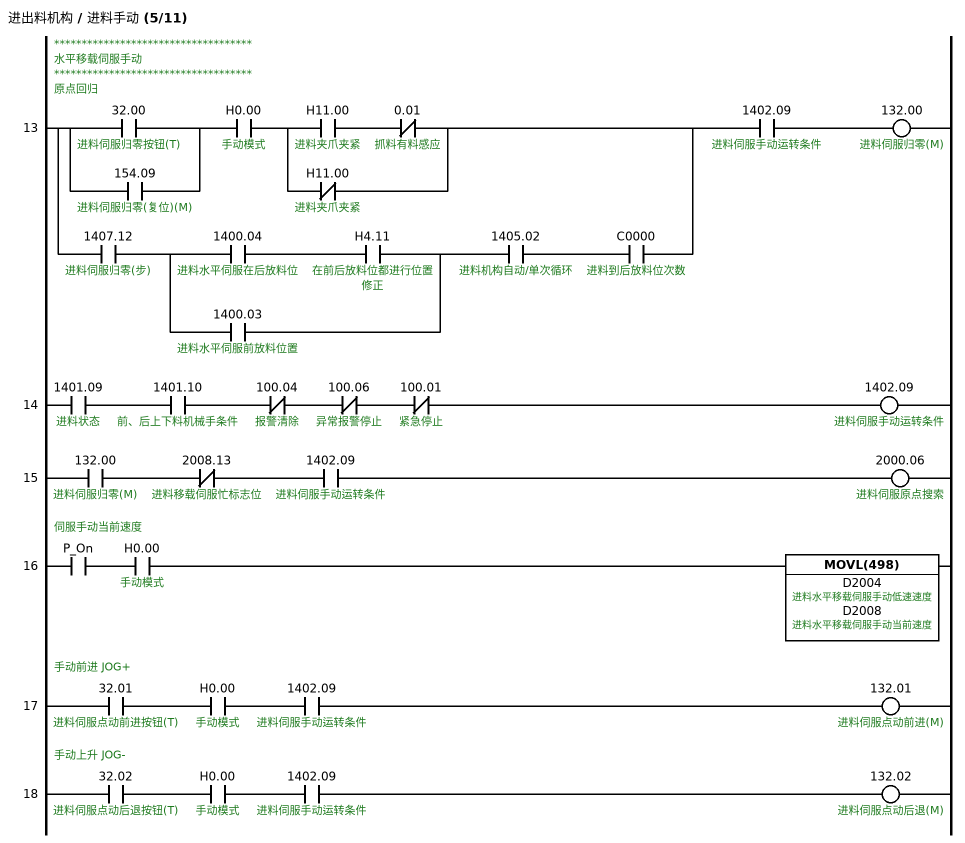
; [picture p72: 进出料机构 / 进料手动, rungs 13-18]
; rung 13: ************************************ / 水平移载伺服手动 / ************************************ / 原点回归
LD 32.00  ; 进料伺服归零按钮(T)
OR 154.09  ; 进料伺服归零(复位)(M)
AND H0.00  ; 手动模式
LD H11.00  ; 进料夹爪夹紧
ANDNOT 0.01  ; 抓料有料感应
ORNOT H11.00  ; 进料夹爪夹紧
ANDLD
LD 1407.12  ; 进料伺服归零(步)
LD 1400.04  ; 进料水平伺服在后放料位
AND H4.11  ; 在前后放料位都进行位置修正
OR 1400.03  ; 进料水平伺服前放料位置
ANDLD
AND 1405.02  ; 进料机构自动/单次循环
AND C0000  ; 进料到后放料位次数
ORLD
AND 1402.09  ; 进料伺服手动运转条件
OUT 132.00  ; 进料伺服归零(M)
; rung 14
LD 1401.09  ; 进料状态
AND 1401.10  ; 前、后上下料机械手条件
ANDNOT 100.04  ; 报警清除
ANDNOT 100.06  ; 异常报警停止
ANDNOT 100.01  ; 紧急停止
OUT 1402.09  ; 进料伺服手动运转条件
; rung 15
LD 132.00  ; 进料伺服归零(M)
ANDNOT 2008.13  ; 进料移载伺服忙标志位
AND 1402.09  ; 进料伺服手动运转条件
OUT 2000.06  ; 进料伺服原点搜索
; rung 16: 伺服手动当前速度
LD P_On
AND H0.00  ; 手动模式
MOVL(498) D2004 D2008  ; 进料水平移载伺服手动低速速度, 进料水平移载伺服手动当前速度
; rung 17: 手动前进 JOG+
LD 32.01  ; 进料伺服点动前进按钮(T)
AND H0.00  ; 手动模式
AND 1402.09  ; 进料伺服手动运转条件
OUT 132.01  ; 进料伺服点动前进(M)
; rung 18: 手动上升 JOG-
LD 32.02  ; 进料伺服点动后退按钮(T)
AND H0.00  ; 手动模式
AND 1402.09  ; 进料伺服手动运转条件
OUT 132.02  ; 进料伺服点动后退(M)

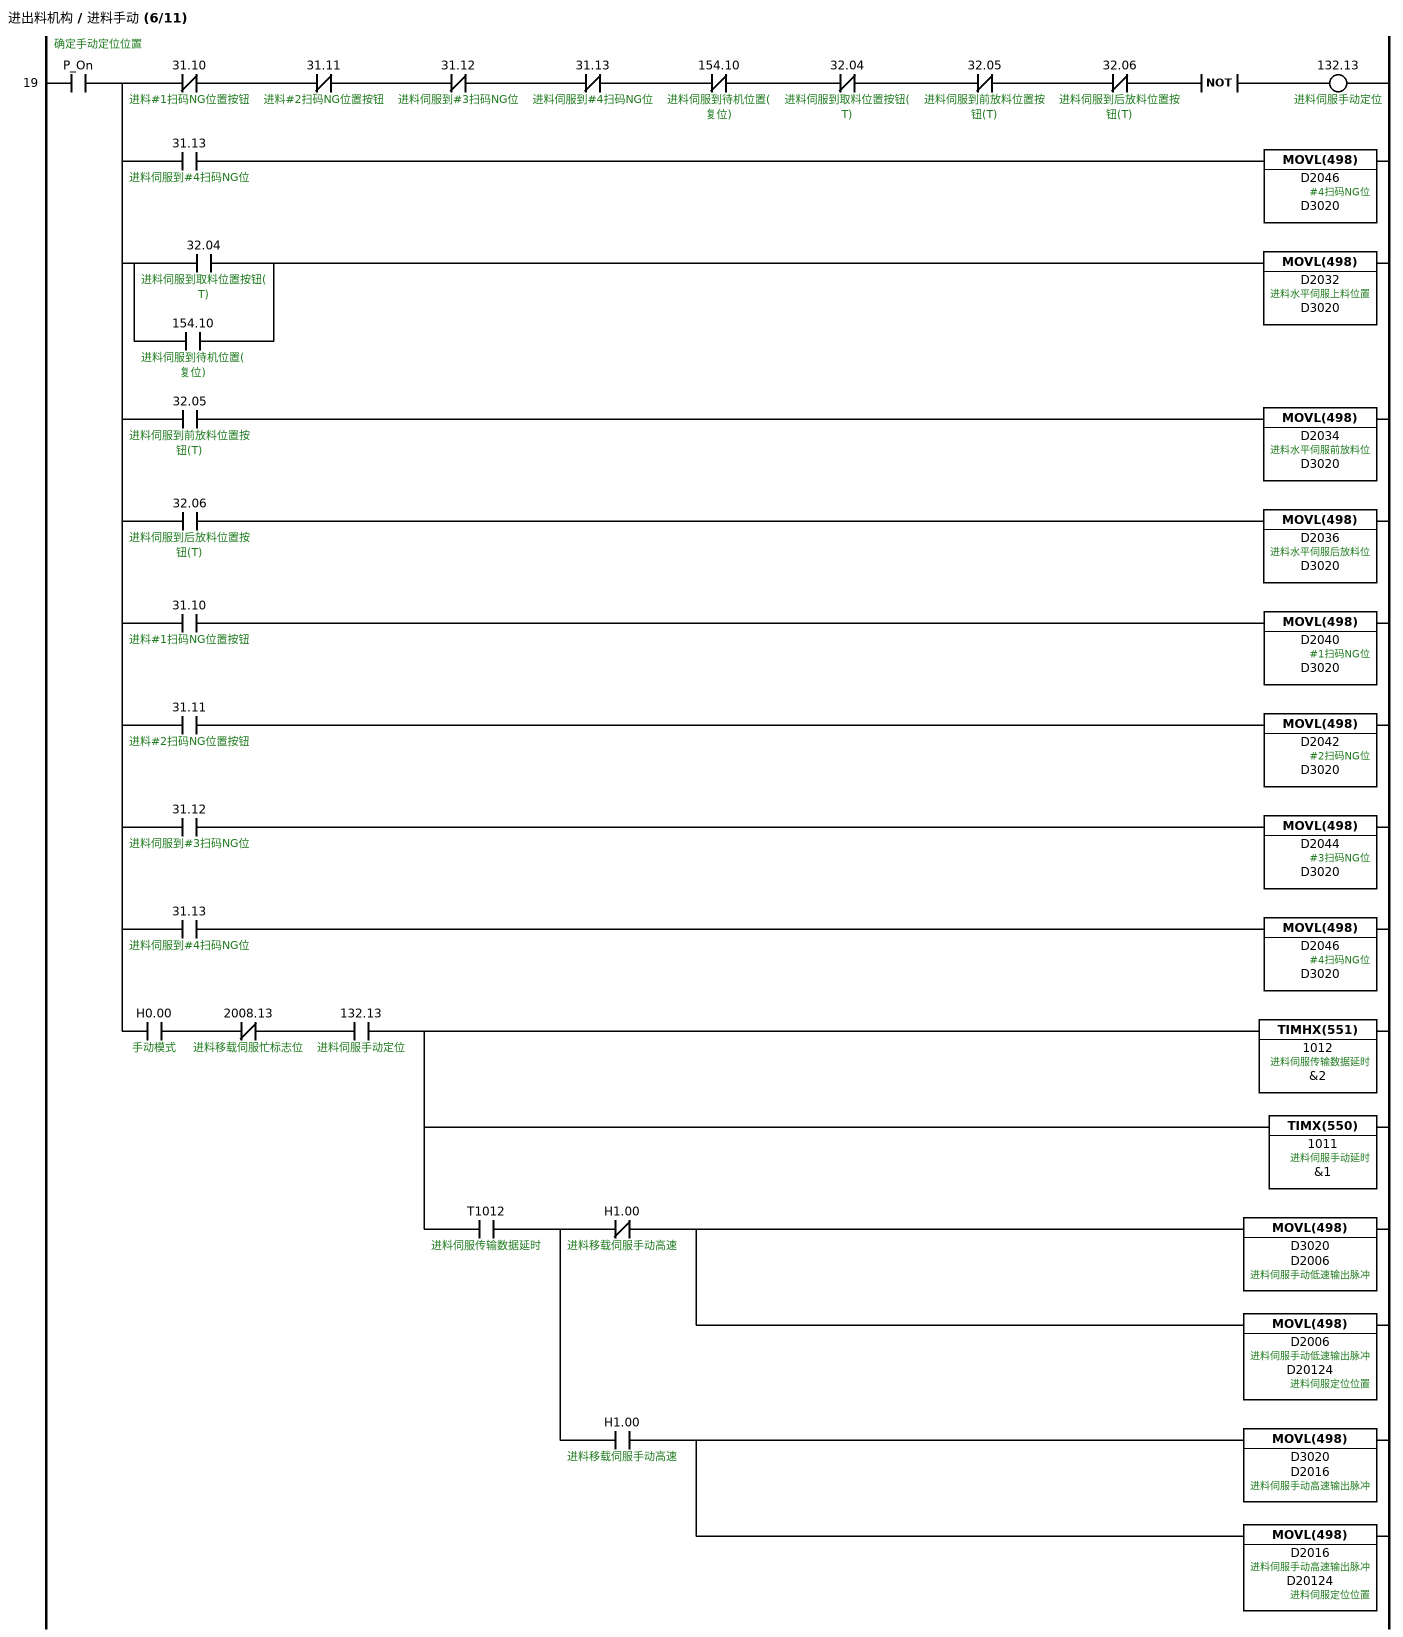
; rung 19: 确定手动定位位置
LD P_On
OUT TR0
ANDNOT 31.10  ; 进料#1扫码NG位置按钮
ANDNOT 31.11  ; 进料#2扫码NG位置按钮
ANDNOT 31.12  ; 进料伺服到#3扫码NG位
ANDNOT 31.13  ; 进料伺服到#4扫码NG位
ANDNOT 154.10  ; 进料伺服到待机位置(复位)
ANDNOT 32.04  ; 进料伺服到取料位置按钮(T)
ANDNOT 32.05  ; 进料伺服到前放料位置按钮(T)
ANDNOT 32.06  ; 进料伺服到后放料位置按钮(T)
NOT(520)
OUT 132.13  ; 进料伺服手动定位
LD TR0
AND 31.13  ; 进料伺服到#4扫码NG位
MOVL(498) D2046 D3020  ; #4扫码NG位
LD TR0
LD 32.04  ; 进料伺服到取料位置按钮(T)
OR 154.10  ; 进料伺服到待机位置(复位)
ANDLD
MOVL(498) D2032 D3020  ; 进料水平伺服上料位置
LD TR0
AND 32.05  ; 进料伺服到前放料位置按钮(T)
MOVL(498) D2034 D3020  ; 进料水平伺服前放料位
LD TR0
AND 32.06  ; 进料伺服到后放料位置按钮(T)
MOVL(498) D2036 D3020  ; 进料水平伺服后放料位
LD TR0
AND 31.10  ; 进料#1扫码NG位置按钮
MOVL(498) D2040 D3020  ; #1扫码NG位
LD TR0
AND 31.11  ; 进料#2扫码NG位置按钮
MOVL(498) D2042 D3020  ; #2扫码NG位
LD TR0
AND 31.12  ; 进料伺服到#3扫码NG位
MOVL(498) D2044 D3020  ; #3扫码NG位
LD TR0
AND 31.13  ; 进料伺服到#4扫码NG位
MOVL(498) D2046 D3020  ; #4扫码NG位
LD TR0
AND H0.00  ; 手动模式
ANDNOT 2008.13  ; 进料移载伺服忙标志位
AND 132.13  ; 进料伺服手动定位
TIMHX(551) 1012 &2  ; 进料伺服传输数据延时
TIMX(550) 1011 &1  ; 进料伺服手动延时
AND T1012  ; 进料伺服传输数据延时
OUT TR0
ANDNOT H1.00  ; 进料移载伺服手动高速
MOVL(498) D3020 D2006  ; 进料伺服手动低速输出脉冲
MOVL(498) D2006 D20124  ; 进料伺服手动低速输出脉冲, 进料伺服定位位置
LD TR0
AND H1.00  ; 进料移载伺服手动高速
MOVL(498) D3020 D2016  ; 进料伺服手动高速输出脉冲
MOVL(498) D2016 D20124  ; 进料伺服手动高速输出脉冲, 进料伺服定位位置

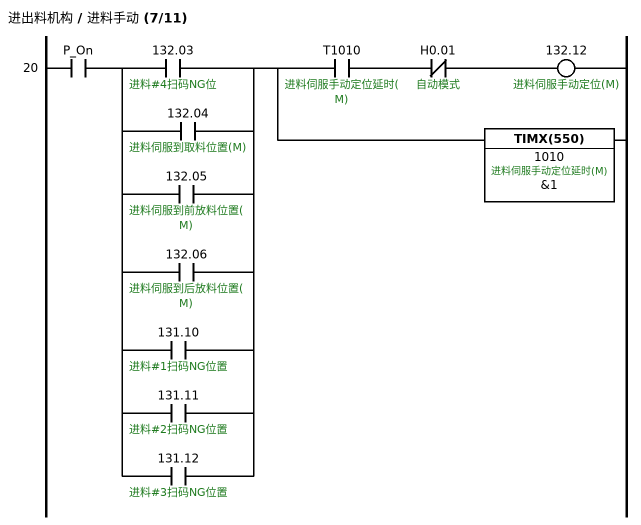
; rung 20
LD P_On
LD 132.03  ; 进料#4扫码NG位
OR 132.04  ; 进料伺服到取料位置(M)
OR 132.05  ; 进料伺服到前放料位置(M)
OR 132.06  ; 进料伺服到后放料位置(M)
OR 131.10  ; 进料#1扫码NG位置
OR 131.11  ; 进料#2扫码NG位置
OR 131.12  ; 进料#3扫码NG位置
ANDLD
OUT TR0
AND T1010  ; 进料伺服手动定位延时(M)
ANDNOT H0.01  ; 自动模式
OUT 132.12  ; 进料伺服手动定位(M)
LD TR0
TIMX(550) 1010 &1  ; 进料伺服手动定位延时(M)

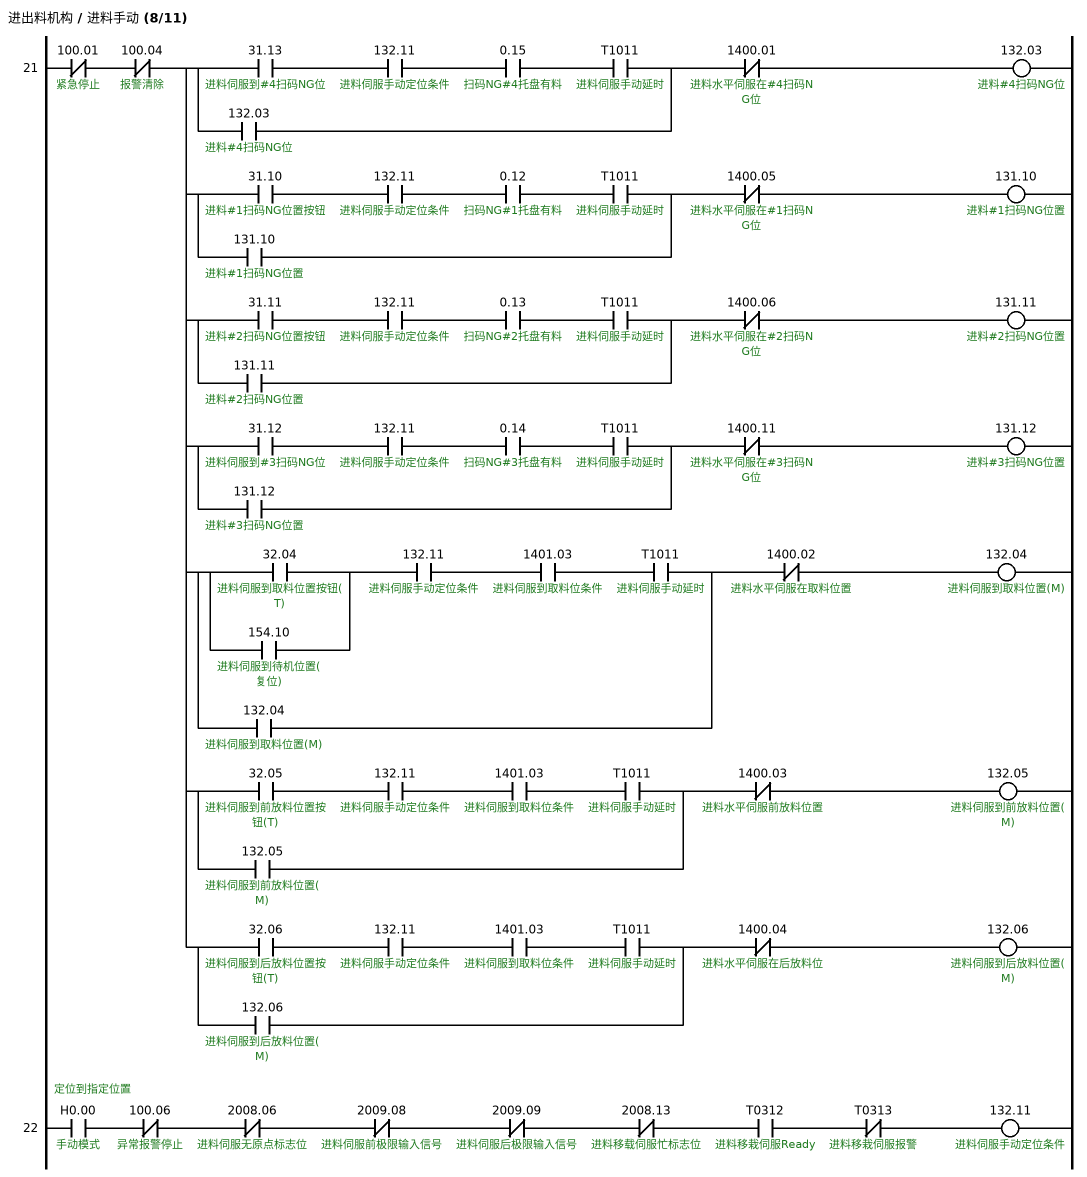
; rung 21
LDNOT 100.01  ; 紧急停止
ANDNOT 100.04  ; 报警清除
OUT TR0
LD 31.13  ; 进料伺服到#4扫码NG位
AND 132.11  ; 进料伺服手动定位条件
AND 0.15  ; 扫码NG#4托盘有料
AND T1011  ; 进料伺服手动延时
OR 132.03  ; 进料#4扫码NG位
ANDLD
ANDNOT 1400.01  ; 进料水平伺服在#4扫码NG位
OUT 132.03  ; 进料#4扫码NG位
LD TR0
LD 31.10  ; 进料#1扫码NG位置按钮
AND 132.11  ; 进料伺服手动定位条件
AND 0.12  ; 扫码NG#1托盘有料
AND T1011  ; 进料伺服手动延时
OR 131.10  ; 进料#1扫码NG位置
ANDLD
ANDNOT 1400.05  ; 进料水平伺服在#1扫码NG位
OUT 131.10  ; 进料#1扫码NG位置
LD TR0
LD 31.11  ; 进料#2扫码NG位置按钮
AND 132.11  ; 进料伺服手动定位条件
AND 0.13  ; 扫码NG#2托盘有料
AND T1011  ; 进料伺服手动延时
OR 131.11  ; 进料#2扫码NG位置
ANDLD
ANDNOT 1400.06  ; 进料水平伺服在#2扫码NG位
OUT 131.11  ; 进料#2扫码NG位置
LD TR0
LD 31.12  ; 进料伺服到#3扫码NG位
AND 132.11  ; 进料伺服手动定位条件
AND 0.14  ; 扫码NG#3托盘有料
AND T1011  ; 进料伺服手动延时
OR 131.12  ; 进料#3扫码NG位置
ANDLD
ANDNOT 1400.11  ; 进料水平伺服在#3扫码NG位
OUT 131.12  ; 进料#3扫码NG位置
LD TR0
LD 32.04  ; 进料伺服到取料位置按钮(T)
OR 154.10  ; 进料伺服到待机位置(复位)
AND 132.11  ; 进料伺服手动定位条件
AND 1401.03  ; 进料伺服到取料位条件
AND T1011  ; 进料伺服手动延时
OR 132.04  ; 进料伺服到取料位置(M)
ANDLD
ANDNOT 1400.02  ; 进料水平伺服在取料位置
OUT 132.04  ; 进料伺服到取料位置(M)
LD TR0
LD 32.05  ; 进料伺服到前放料位置按钮(T)
AND 132.11  ; 进料伺服手动定位条件
AND 1401.03  ; 进料伺服到取料位条件
AND T1011  ; 进料伺服手动延时
OR 132.05  ; 进料伺服到前放料位置(M)
ANDLD
ANDNOT 1400.03  ; 进料水平伺服前放料位置
OUT 132.05  ; 进料伺服到前放料位置(M)
LD TR0
LD 32.06  ; 进料伺服到后放料位置按钮(T)
AND 132.11  ; 进料伺服手动定位条件
AND 1401.03  ; 进料伺服到取料位条件
AND T1011  ; 进料伺服手动延时
OR 132.06  ; 进料伺服到后放料位置(M)
ANDLD
ANDNOT 1400.04  ; 进料水平伺服在后放料位
OUT 132.06  ; 进料伺服到后放料位置(M)
; rung 22: 定位到指定位置
LD H0.00  ; 手动模式
ANDNOT 100.06  ; 异常报警停止
ANDNOT 2008.06  ; 进料伺服无原点标志位
ANDNOT 2009.08  ; 进料伺服前极限输入信号
ANDNOT 2009.09  ; 进料伺服后极限输入信号
ANDNOT 2008.13  ; 进料移载伺服忙标志位
AND T0312  ; 进料移栽伺服Ready
ANDNOT T0313  ; 进料移栽伺服报警
OUT 132.11  ; 进料伺服手动定位条件

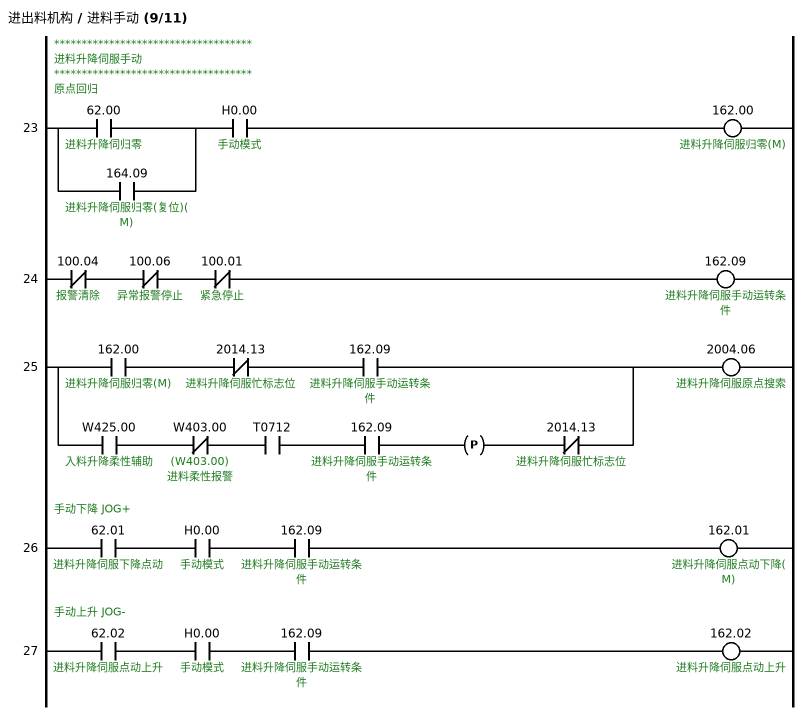
; rung 23: ************************************ / 进料升降伺服手动 / ************************************ / 原点回归
LD 62.00  ; 进料升降伺归零
OR 164.09  ; 进料升降伺服归零(复位)(M)
AND H0.00  ; 手动模式
OUT 162.00  ; 进料升降伺服归零(M)
; rung 24
LDNOT 100.04  ; 报警清除
ANDNOT 100.06  ; 异常报警停止
ANDNOT 100.01  ; 紧急停止
OUT 162.09  ; 进料升降伺服手动运转条件
; rung 25
LD 162.00  ; 进料升降伺服归零(M)
ANDNOT 2014.13  ; 进料升降伺服忙标志位
AND 162.09  ; 进料升降伺服手动运转条件
LD W425.00  ; 入料升降柔性辅助
ANDNOT W403.00  ; (W403.00) 进料柔性报警
AND T0712
AND 162.09  ; 进料升降伺服手动运转条件
UP(521)
ANDNOT 2014.13  ; 进料升降伺服忙标志位
ORLD
OUT 2004.06  ; 进料升降伺服原点搜索
; rung 26: 手动下降 JOG+
LD 62.01  ; 进料升降伺服下降点动
AND H0.00  ; 手动模式
AND 162.09  ; 进料升降伺服手动运转条件
OUT 162.01  ; 进料升降伺服点动下降(M)
; rung 27: 手动上升 JOG-
LD 62.02  ; 进料升降伺服点动上升
AND H0.00  ; 手动模式
AND 162.09  ; 进料升降伺服手动运转条件
OUT 162.02  ; 进料升降伺服点动上升

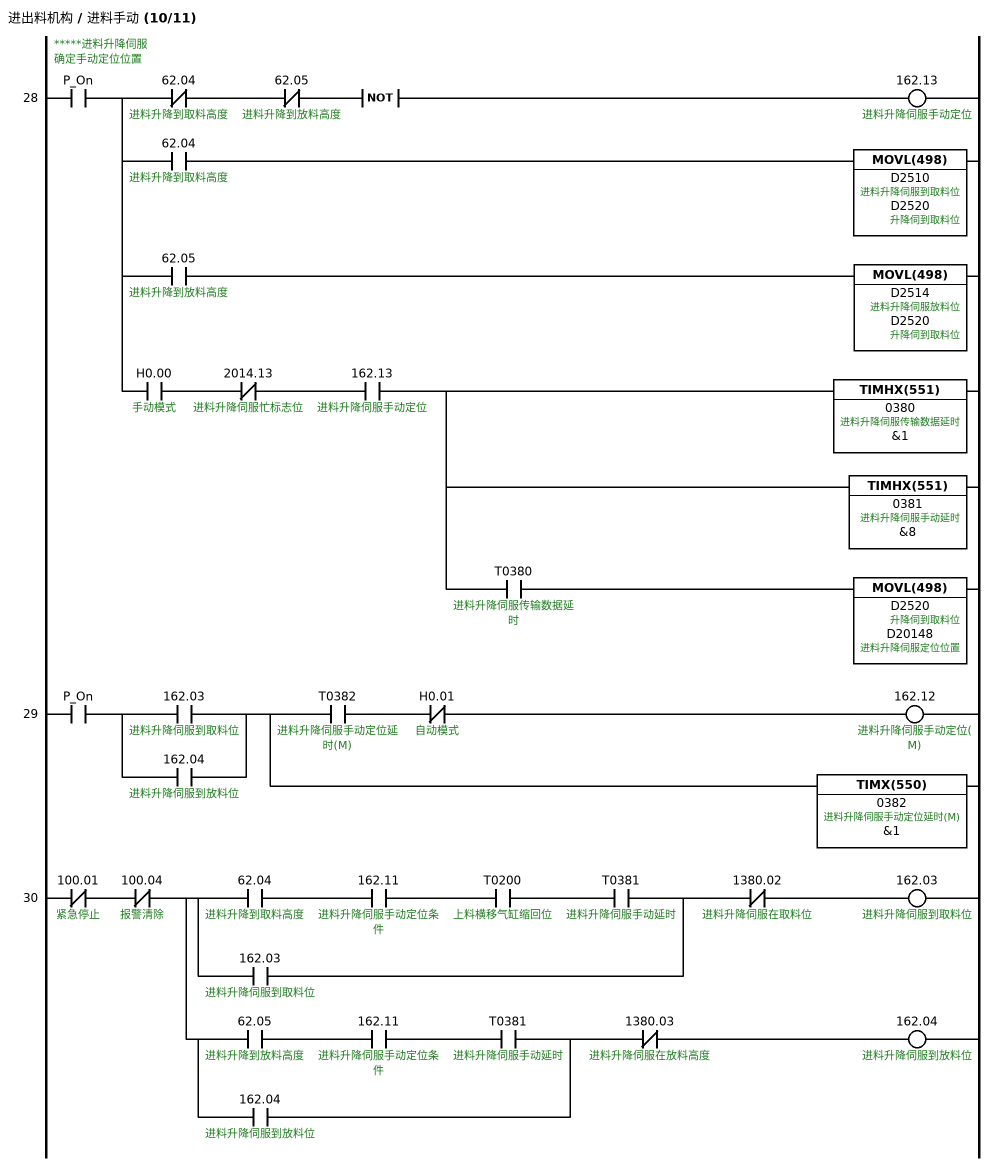
; rung 28: *****进料升降伺服 / 确定手动定位位置
LD P_On
OUT TR0
ANDNOT 62.04  ; 进料升降到取料高度
ANDNOT 62.05  ; 进料升降到放料高度
NOT(520)
OUT 162.13  ; 进料升降伺服手动定位
LD TR0
AND 62.04  ; 进料升降到取料高度
MOVL(498) D2510 D2520  ; 进料升降伺服到取料位, 升降伺到取料位
LD TR0
AND 62.05  ; 进料升降到放料高度
MOVL(498) D2514 D2520  ; 进料升降伺服放料位, 升降伺到取料位
LD TR0
AND H0.00  ; 手动模式
ANDNOT 2014.13  ; 进料升降伺服忙标志位
AND 162.13  ; 进料升降伺服手动定位
TIMHX(551) 0380 &1  ; 进料升降伺服传输数据延时
TIMHX(551) 0381 &8  ; 进料升降伺服手动延时
AND T0380  ; 进料升降伺服传输数据延时
MOVL(498) D2520 D20148  ; 升降伺到取料位, 进料升降伺服定位位置
; rung 29
LD P_On
LD 162.03  ; 进料升降伺服到取料位
OR 162.04  ; 进料升降伺服到放料位
ANDLD
OUT TR0
AND T0382  ; 进料升降伺服手动定位延时(M)
ANDNOT H0.01  ; 自动模式
OUT 162.12  ; 进料升降伺服手动定位(M)
LD TR0
TIMX(550) 0382 &1  ; 进料升降伺服手动定位延时(M)
; rung 30
LDNOT 100.01  ; 紧急停止
ANDNOT 100.04  ; 报警清除
OUT TR0
LD 62.04  ; 进料升降到取料高度
AND 162.11  ; 进料升降伺服手动定位条件
AND T0200  ; 上料横移气缸缩回位
AND T0381  ; 进料升降伺服手动延时
OR 162.03  ; 进料升降伺服到取料位
ANDLD
ANDNOT 1380.02  ; 进料升降伺服在取料位
OUT 162.03  ; 进料升降伺服到取料位
LD TR0
LD 62.05  ; 进料升降到放料高度
AND 162.11  ; 进料升降伺服手动定位条件
AND T0381  ; 进料升降伺服手动延时
OR 162.04  ; 进料升降伺服到放料位
ANDLD
ANDNOT 1380.03  ; 进料升降伺服在放料高度
OUT 162.04  ; 进料升降伺服到放料位

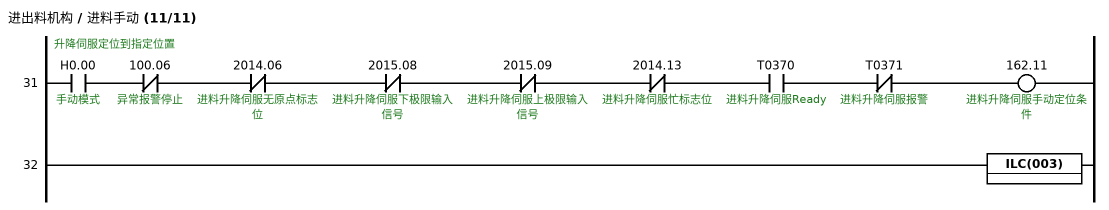
; rung 31: 升降伺服定位到指定位置
LD H0.00  ; 手动模式
ANDNOT 100.06  ; 异常报警停止
ANDNOT 2014.06  ; 进料升降伺服无原点标志位
ANDNOT 2015.08  ; 进料升降伺服下极限输入信号
ANDNOT 2015.09  ; 进料升降伺服上极限输入信号
ANDNOT 2014.13  ; 进料升降伺服忙标志位
AND T0370  ; 进料升降伺服Ready
ANDNOT T0371  ; 进料升降伺服报警
OUT 162.11  ; 进料升降伺服手动定位条件
; rung 32
ILC(003)

### Section 进料自动

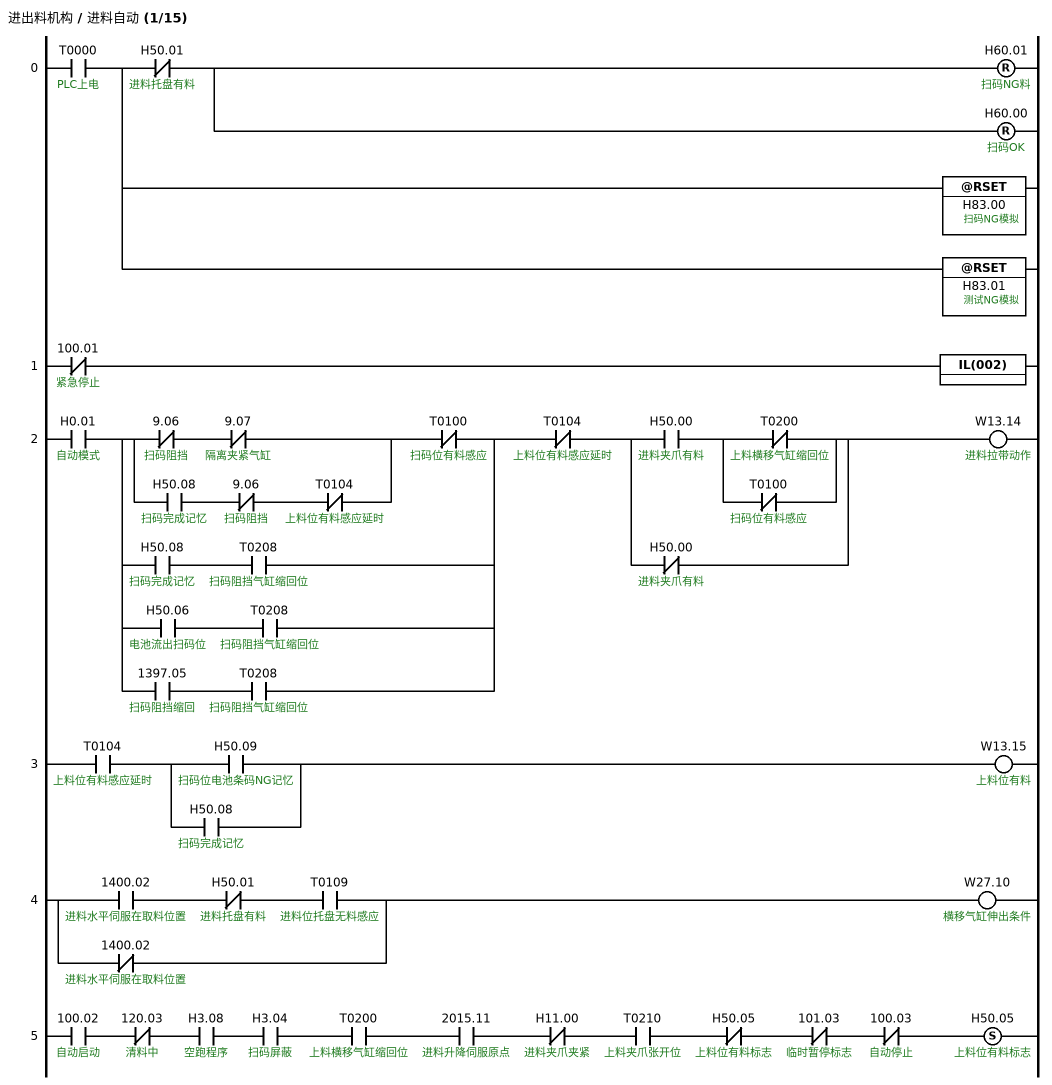
; rung 0
LD T0000  ; PLC上电
OUT TR0
ANDNOT H50.01  ; 进料托盘有料
RSET H60.01  ; 扫码NG料
RSET H60.00  ; 扫码OK
LD TR0
@RSET H83.00  ; 扫码NG模拟
@RSET H83.01  ; 测试NG模拟
; rung 1
LDNOT 100.01  ; 紧急停止
IL(002)
; rung 2
LD H0.01  ; 自动模式
LDNOT 9.06  ; 扫码阻挡
ANDNOT 9.07  ; 隔离夹紧气缸
LD H50.08  ; 扫码完成记忆
ANDNOT 9.06  ; 扫码阻挡
ANDNOT T0104  ; 上料位有料感应延时
ORLD
ANDNOT T0100  ; 扫码位有料感应
LD H50.08  ; 扫码完成记忆
AND T0208  ; 扫码阻挡气缸缩回位
ORLD
LD H50.06  ; 电池流出扫码位
AND T0208  ; 扫码阻挡气缸缩回位
ORLD
LD 1397.05  ; 扫码阻挡缩回
AND T0208  ; 扫码阻挡气缸缩回位
ORLD
ANDLD
ANDNOT T0104  ; 上料位有料感应延时
LD H50.00  ; 进料夹爪有料
LDNOT T0200  ; 上料横移气缸缩回位
ORNOT T0100  ; 扫码位有料感应
ANDLD
ORNOT H50.00  ; 进料夹爪有料
ANDLD
OUT W13.14  ; 进料拉带动作
; rung 3
LD T0104  ; 上料位有料感应延时
LD H50.09  ; 扫码位电池条码NG记忆
OR H50.08  ; 扫码完成记忆
ANDLD
OUT W13.15  ; 上料位有料
; rung 4
LD 1400.02  ; 进料水平伺服在取料位置
ANDNOT H50.01  ; 进料托盘有料
AND T0109  ; 进料位托盘无料感应
ORNOT 1400.02  ; 进料水平伺服在取料位置
OUT W27.10  ; 横移气缸伸出条件
; rung 5
LD 100.02  ; 自动启动
ANDNOT 120.03  ; 清料中
AND H3.08  ; 空跑程序
AND H3.04  ; 扫码屏蔽
AND T0200  ; 上料横移气缸缩回位
AND 2015.11  ; 进料升降伺服原点
ANDNOT H11.00  ; 进料夹爪夹紧
AND T0210  ; 上料夹爪张开位
ANDNOT H50.05  ; 上料位有料标志
ANDNOT 101.03  ; 临时暂停标志
ANDNOT 100.03  ; 自动停止
SET H50.05  ; 上料位有料标志

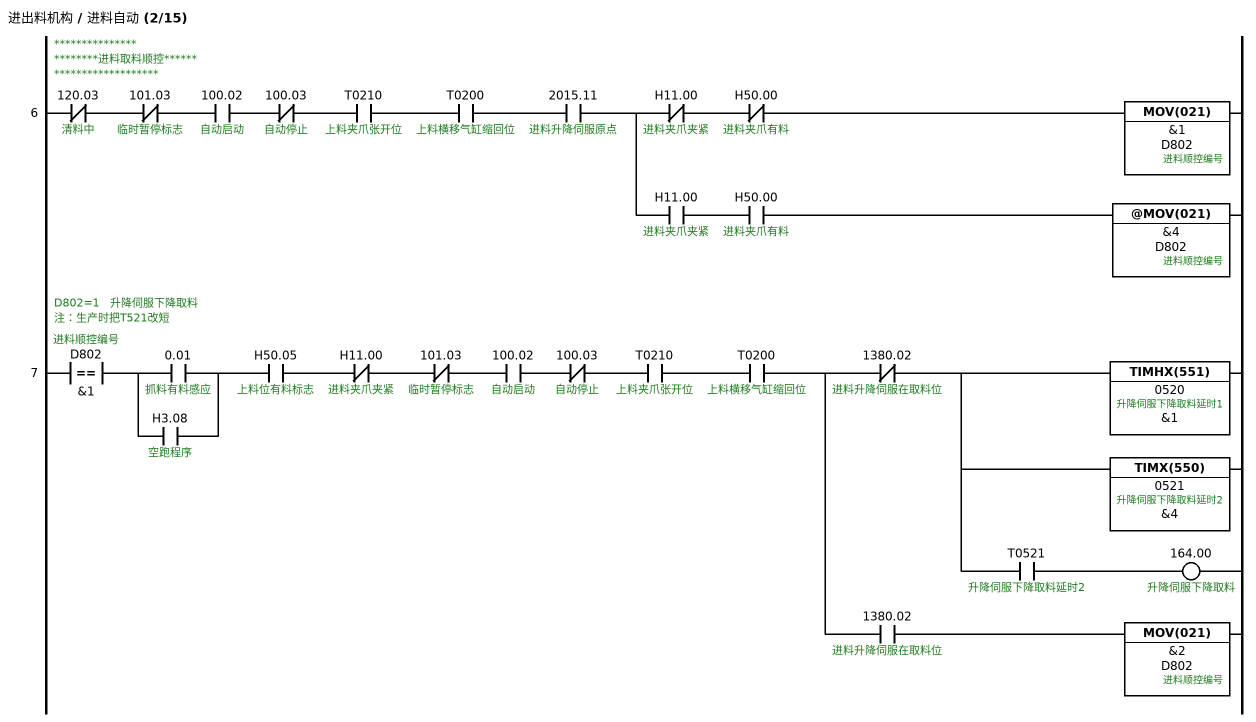
; rung 6: *************** / ********进料取料顺控****** / *******************
LDNOT 120.03  ; 清料中
ANDNOT 101.03  ; 临时暂停标志
AND 100.02  ; 自动启动
ANDNOT 100.03  ; 自动停止
AND T0210  ; 上料夹爪张开位
AND T0200  ; 上料横移气缸缩回位
AND 2015.11  ; 进料升降伺服原点
OUT TR0
ANDNOT H11.00  ; 进料夹爪夹紧
ANDNOT H50.00  ; 进料夹爪有料
MOV(021) &1 D802  ; 进料顺控编号
LD TR0
AND H11.00  ; 进料夹爪夹紧
AND H50.00  ; 进料夹爪有料
@MOV(021) &4 D802  ; 进料顺控编号
; rung 7: D802=1   升降伺服下降取料 / 注：生产时把T521改短
LD=(300) D802 &1  ; 进料顺控编号
LD 0.01  ; 抓料有料感应
OR H3.08  ; 空跑程序
ANDLD
AND H50.05  ; 上料位有料标志
ANDNOT H11.00  ; 进料夹爪夹紧
ANDNOT 101.03  ; 临时暂停标志
AND 100.02  ; 自动启动
ANDNOT 100.03  ; 自动停止
AND T0210  ; 上料夹爪张开位
AND T0200  ; 上料横移气缸缩回位
OUT TR0
ANDNOT 1380.02  ; 进料升降伺服在取料位
TIMHX(551) 0520 &1  ; 升降伺服下降取料延时1
TIMX(550) 0521 &4  ; 升降伺服下降取料延时2
AND T0521  ; 升降伺服下降取料延时2
OUT 164.00  ; 升降伺服下降取料
LD TR0
AND 1380.02  ; 进料升降伺服在取料位
MOV(021) &2 D802  ; 进料顺控编号

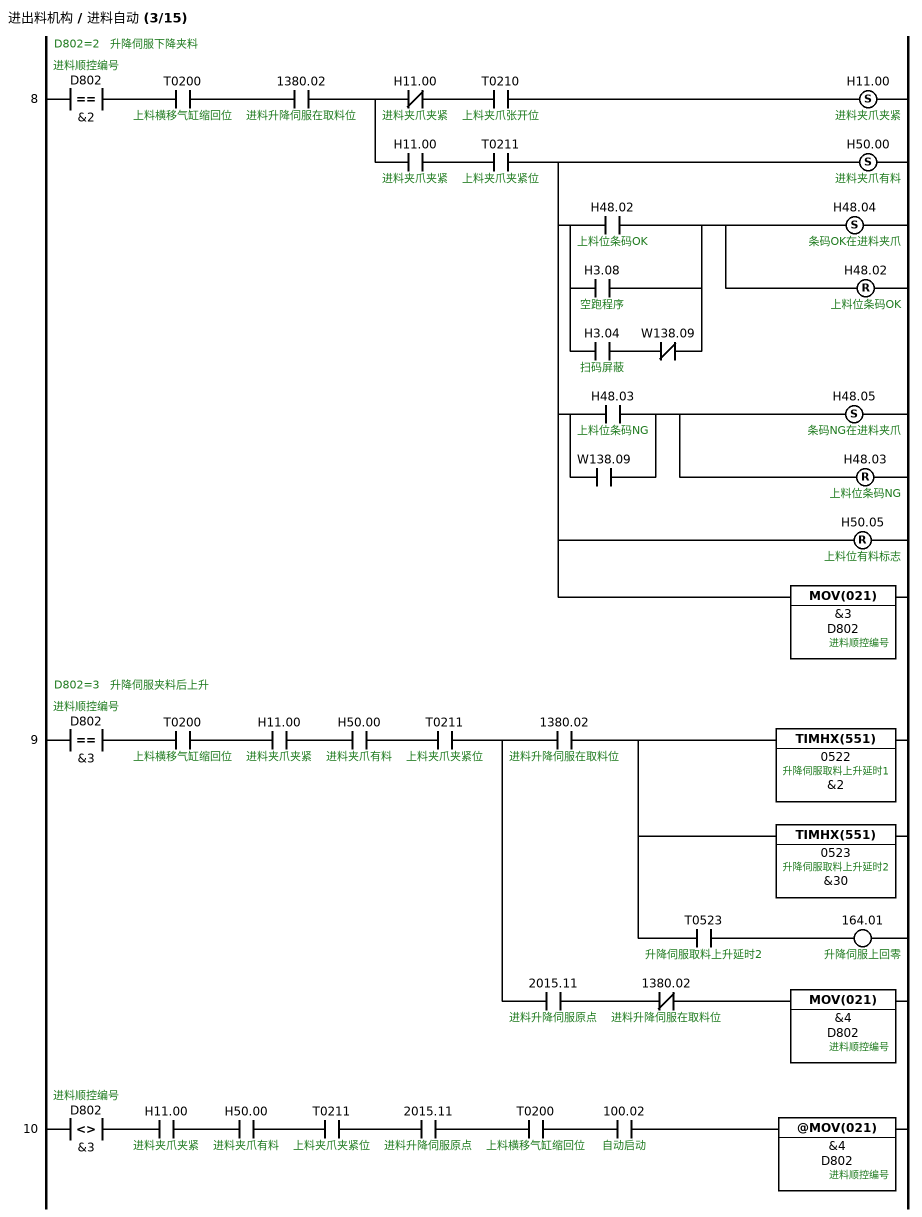
; rung 8: D802=2   升降伺服下降夹料
LD=(300) D802 &2  ; 进料顺控编号
AND T0200  ; 上料横移气缸缩回位
AND 1380.02  ; 进料升降伺服在取料位
OUT TR0
ANDNOT H11.00  ; 进料夹爪夹紧
AND T0210  ; 上料夹爪张开位
SET H11.00  ; 进料夹爪夹紧
LD TR0
AND H11.00  ; 进料夹爪夹紧
AND T0211  ; 上料夹爪夹紧位
OUT TR0
SET H50.00  ; 进料夹爪有料
LD H48.02  ; 上料位条码OK
OR H3.08  ; 空跑程序
LD H3.04  ; 扫码屏蔽
ANDNOT W138.09
ORLD
ANDLD
SET H48.04  ; 条码OK在进料夹爪
RSET H48.02  ; 上料位条码OK
LD TR0
LD H48.03  ; 上料位条码NG
OR W138.09
ANDLD
SET H48.05  ; 条码NG在进料夹爪
RSET H48.03  ; 上料位条码NG
LD TR0
RSET H50.05  ; 上料位有料标志
MOV(021) &3 D802  ; 进料顺控编号
; rung 9: D802=3   升降伺服夹料后上升
LD=(300) D802 &3  ; 进料顺控编号
AND T0200  ; 上料横移气缸缩回位
AND H11.00  ; 进料夹爪夹紧
AND H50.00  ; 进料夹爪有料
AND T0211  ; 上料夹爪夹紧位
OUT TR0
AND 1380.02  ; 进料升降伺服在取料位
TIMHX(551) 0522 &2  ; 升降伺服取料上升延时1
TIMHX(551) 0523 &30  ; 升降伺服取料上升延时2
AND T0523  ; 升降伺服取料上升延时2
OUT 164.01  ; 升降伺服上回零
LD TR0
AND 2015.11  ; 进料升降伺服原点
ANDNOT 1380.02  ; 进料升降伺服在取料位
MOV(021) &4 D802  ; 进料顺控编号
; rung 10
LD<>(305) D802 &3  ; 进料顺控编号
AND H11.00  ; 进料夹爪夹紧
AND H50.00  ; 进料夹爪有料
AND T0211  ; 上料夹爪夹紧位
AND 2015.11  ; 进料升降伺服原点
AND T0200  ; 上料横移气缸缩回位
AND 100.02  ; 自动启动
@MOV(021) &4 D802  ; 进料顺控编号

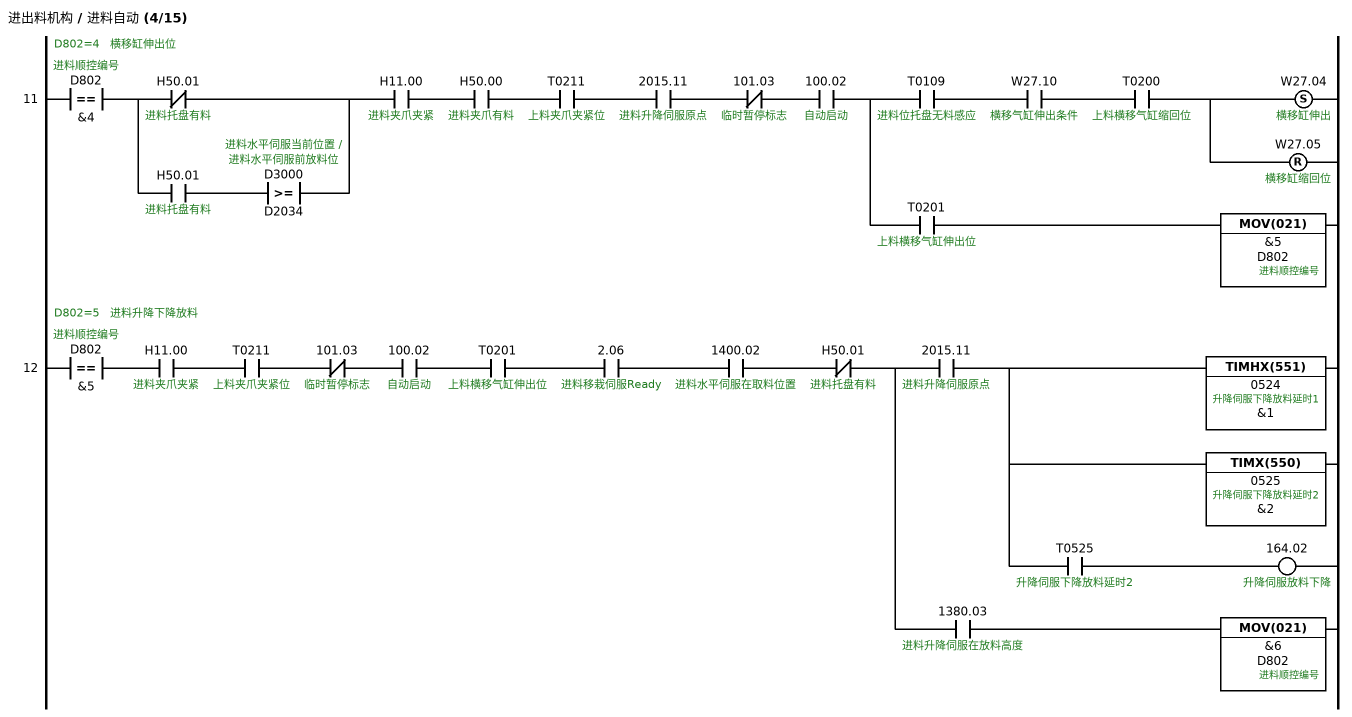
; rung 11: D802=4   横移缸伸出位
LD=(300) D802 &4  ; 进料顺控编号
LDNOT H50.01  ; 进料托盘有料
LD H50.01  ; 进料托盘有料
AND>=SL(328) D3000 D2034  ; 进料水平伺服当前位置, 进料水平伺服前放料位
ORLD
ANDLD
AND H11.00  ; 进料夹爪夹紧
AND H50.00  ; 进料夹爪有料
AND T0211  ; 上料夹爪夹紧位
AND 2015.11  ; 进料升降伺服原点
ANDNOT 101.03  ; 临时暂停标志
AND 100.02  ; 自动启动
OUT TR0
AND T0109  ; 进料位托盘无料感应
AND W27.10  ; 横移气缸伸出条件
AND T0200  ; 上料横移气缸缩回位
SET W27.04  ; 横移缸伸出
RSET W27.05  ; 横移缸缩回位
LD TR0
AND T0201  ; 上料横移气缸伸出位
MOV(021) &5 D802  ; 进料顺控编号
; rung 12: D802=5   进料升降下降放料
LD=(300) D802 &5  ; 进料顺控编号
AND H11.00  ; 进料夹爪夹紧
AND T0211  ; 上料夹爪夹紧位
ANDNOT 101.03  ; 临时暂停标志
AND 100.02  ; 自动启动
AND T0201  ; 上料横移气缸伸出位
AND 2.06  ; 进料移栽伺服Ready
AND 1400.02  ; 进料水平伺服在取料位置
ANDNOT H50.01  ; 进料托盘有料
OUT TR0
AND 2015.11  ; 进料升降伺服原点
TIMHX(551) 0524 &1  ; 升降伺服下降放料延时1
TIMX(550) 0525 &2  ; 升降伺服下降放料延时2
AND T0525  ; 升降伺服下降放料延时2
OUT 164.02  ; 升降伺服放料下降
LD TR0
AND 1380.03  ; 进料升降伺服在放料高度
MOV(021) &6 D802  ; 进料顺控编号

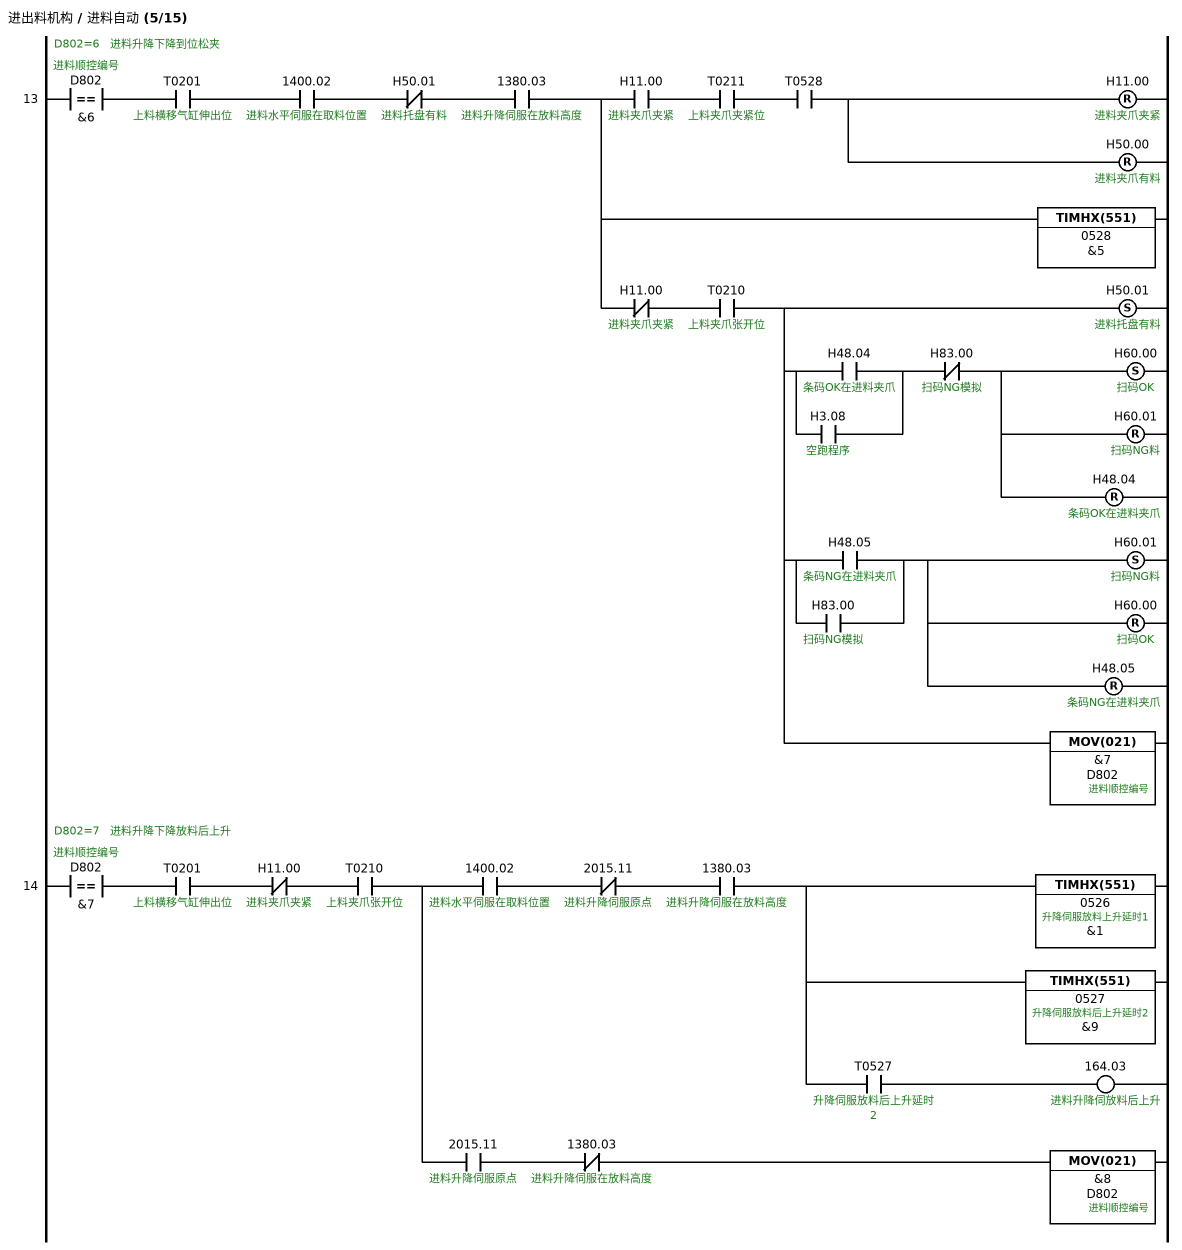
; rung 13: D802=6   进料升降下降到位松夹
LD=(300) D802 &6  ; 进料顺控编号
AND T0201  ; 上料横移气缸伸出位
AND 1400.02  ; 进料水平伺服在取料位置
ANDNOT H50.01  ; 进料托盘有料
AND 1380.03  ; 进料升降伺服在放料高度
OUT TR0
AND H11.00  ; 进料夹爪夹紧
AND T0211  ; 上料夹爪夹紧位
AND T0528
RSET H11.00  ; 进料夹爪夹紧
RSET H50.00  ; 进料夹爪有料
LD TR0
TIMHX(551) 0528 &5
ANDNOT H11.00  ; 进料夹爪夹紧
AND T0210  ; 上料夹爪张开位
OUT TR0
SET H50.01  ; 进料托盘有料
LD H48.04  ; 条码OK在进料夹爪
OR H3.08  ; 空跑程序
ANDLD
ANDNOT H83.00  ; 扫码NG模拟
SET H60.00  ; 扫码OK
RSET H60.01  ; 扫码NG料
RSET H48.04  ; 条码OK在进料夹爪
LD TR0
LD H48.05  ; 条码NG在进料夹爪
OR H83.00  ; 扫码NG模拟
ANDLD
SET H60.01  ; 扫码NG料
RSET H60.00  ; 扫码OK
RSET H48.05  ; 条码NG在进料夹爪
LD TR0
MOV(021) &7 D802  ; 进料顺控编号
; rung 14: D802=7   进料升降下降放料后上升
LD=(300) D802 &7  ; 进料顺控编号
AND T0201  ; 上料横移气缸伸出位
ANDNOT H11.00  ; 进料夹爪夹紧
AND T0210  ; 上料夹爪张开位
OUT TR0
AND 1400.02  ; 进料水平伺服在取料位置
ANDNOT 2015.11  ; 进料升降伺服原点
AND 1380.03  ; 进料升降伺服在放料高度
TIMHX(551) 0526 &1  ; 升降伺服放料上升延时1
TIMHX(551) 0527 &9  ; 升降伺服放料后上升延时2
AND T0527  ; 升降伺服放料后上升延时2
OUT 164.03  ; 进料升降伺放料后上升
LD TR0
AND 2015.11  ; 进料升降伺服原点
ANDNOT 1380.03  ; 进料升降伺服在放料高度
MOV(021) &8 D802  ; 进料顺控编号

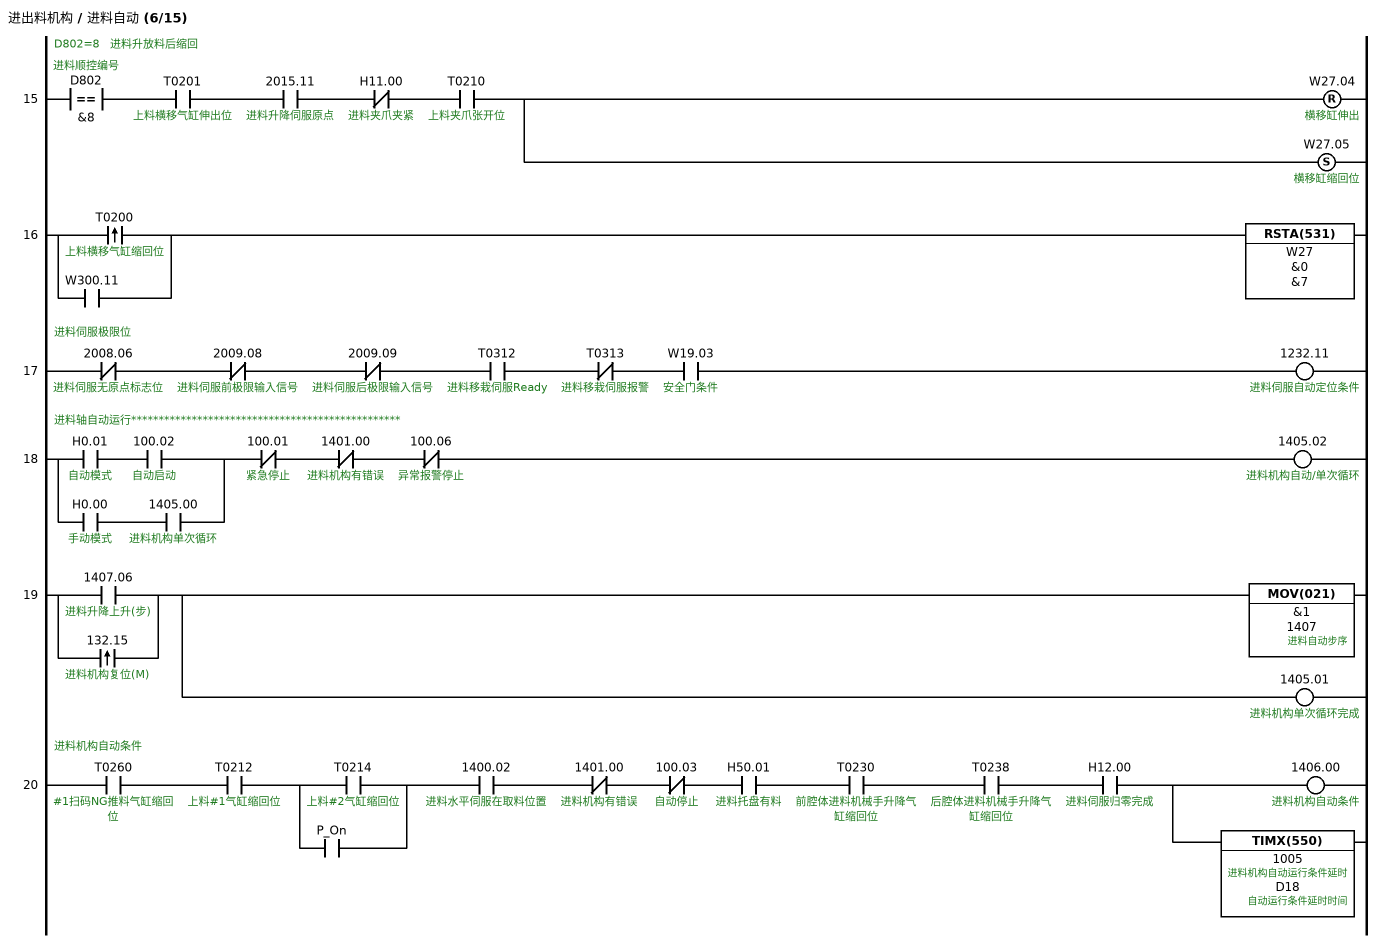
; rung 15: D802=8   进料升放料后缩回
LD=(300) D802 &8  ; 进料顺控编号
AND T0201  ; 上料横移气缸伸出位
AND 2015.11  ; 进料升降伺服原点
ANDNOT H11.00  ; 进料夹爪夹紧
AND T0210  ; 上料夹爪张开位
RSET W27.04  ; 横移缸伸出
SET W27.05  ; 横移缸缩回位
; rung 16
@LD T0200  ; 上料横移气缸缩回位
OR W300.11
RSTA(531) W27 &0 &7
; rung 17: 进料伺服极限位
LDNOT 2008.06  ; 进料伺服无原点标志位
ANDNOT 2009.08  ; 进料伺服前极限输入信号
ANDNOT 2009.09  ; 进料伺服后极限输入信号
AND T0312  ; 进料移栽伺服Ready
ANDNOT T0313  ; 进料移栽伺服报警
AND W19.03  ; 安全门条件
OUT 1232.11  ; 进料伺服自动定位条件
; rung 18: 进料轴自动运行*************************************************
LD H0.01  ; 自动模式
AND 100.02  ; 自动启动
LD H0.00  ; 手动模式
AND 1405.00  ; 进料机构单次循环
ORLD
ANDNOT 100.01  ; 紧急停止
ANDNOT 1401.00  ; 进料机构有错误
ANDNOT 100.06  ; 异常报警停止
OUT 1405.02  ; 进料机构自动/单次循环
; rung 19
LD 1407.06  ; 进料升降上升(步)
@OR 132.15  ; 进料机构复位(M)
MOV(021) &1 1407  ; 进料自动步序
OUT 1405.01  ; 进料机构单次循环完成
; rung 20: 进料机构自动条件
LD T0260  ; #1扫码NG推料气缸缩回位
AND T0212  ; 上料#1气缸缩回位
LD T0214  ; 上料#2气缸缩回位
OR P_On
ANDLD
AND 1400.02  ; 进料水平伺服在取料位置
ANDNOT 1401.00  ; 进料机构有错误
ANDNOT 100.03  ; 自动停止
AND H50.01  ; 进料托盘有料
AND T0230  ; 前腔体进料机械手升降气缸缩回位
AND T0238  ; 后腔体进料机械手升降气缸缩回位
AND H12.00  ; 进料伺服归零完成
OUT 1406.00  ; 进料机构自动条件
TIMX(550) 1005 D18  ; 自动运行条件延时时间, 进料机构自动运行条件延时

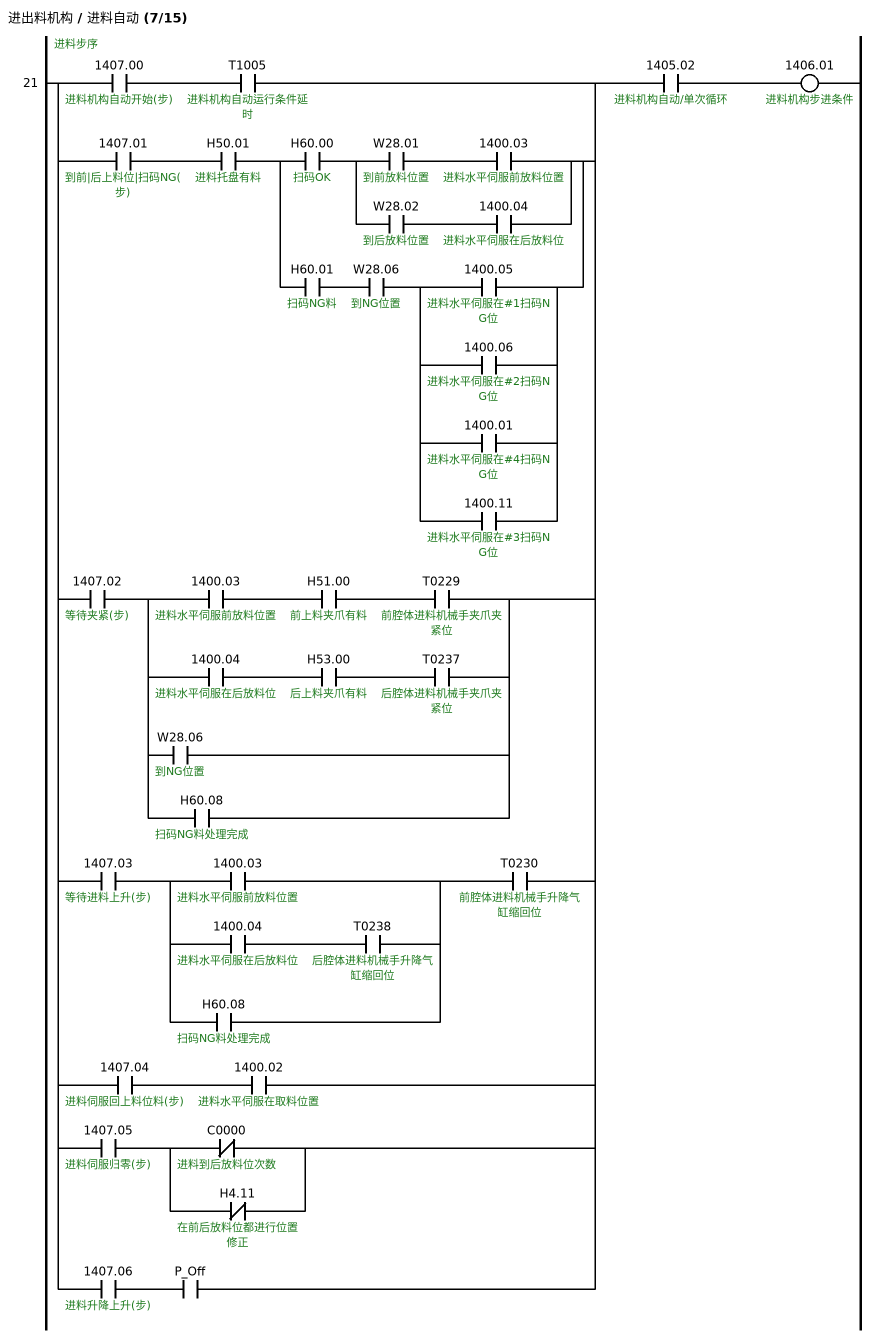
; rung 21: 进料步序
LD 1407.00  ; 进料机构自动开始(步)
AND T1005  ; 进料机构自动运行条件延时
LD 1407.01  ; 到前|后上料位|扫码NG(步)
AND H50.01  ; 进料托盘有料
LD H60.00  ; 扫码OK
LD W28.01  ; 到前放料位置
AND 1400.03  ; 进料水平伺服前放料位置
LD W28.02  ; 到后放料位置
AND 1400.04  ; 进料水平伺服在后放料位
ORLD
ANDLD
LD H60.01  ; 扫码NG料
AND W28.06  ; 到NG位置
LD 1400.05  ; 进料水平伺服在#1扫码NG位
OR 1400.06  ; 进料水平伺服在#2扫码NG位
OR 1400.01  ; 进料水平伺服在#4扫码NG位
OR 1400.11  ; 进料水平伺服在#3扫码NG位
ANDLD
ORLD
ANDLD
ORLD
LD 1407.02  ; 等待夹紧(步)
LD 1400.03  ; 进料水平伺服前放料位置
AND H51.00  ; 前上料夹爪有料
AND T0229  ; 前腔体进料机械手夹爪夹紧位
LD 1400.04  ; 进料水平伺服在后放料位
AND H53.00  ; 后上料夹爪有料
AND T0237  ; 后腔体进料机械手夹爪夹紧位
ORLD
OR W28.06  ; 到NG位置
OR H60.08  ; 扫码NG料处理完成
ANDLD
ORLD
LD 1407.03  ; 等待进料上升(步)
LD 1400.03  ; 进料水平伺服前放料位置
LD 1400.04  ; 进料水平伺服在后放料位
AND T0238  ; 后腔体进料机械手升降气缸缩回位
ORLD
OR H60.08  ; 扫码NG料处理完成
ANDLD
AND T0230  ; 前腔体进料机械手升降气缸缩回位
ORLD
LD 1407.04  ; 进料伺服回上料位料(步)
AND 1400.02  ; 进料水平伺服在取料位置
ORLD
LD 1407.05  ; 进料伺服归零(步)
LDNOT C0000  ; 进料到后放料位次数
ORNOT H4.11  ; 在前后放料位都进行位置修正
ANDLD
ORLD
LD 1407.06  ; 进料升降上升(步)
AND P_Off
ORLD
AND 1405.02  ; 进料机构自动/单次循环
OUT 1406.01  ; 进料机构步进条件

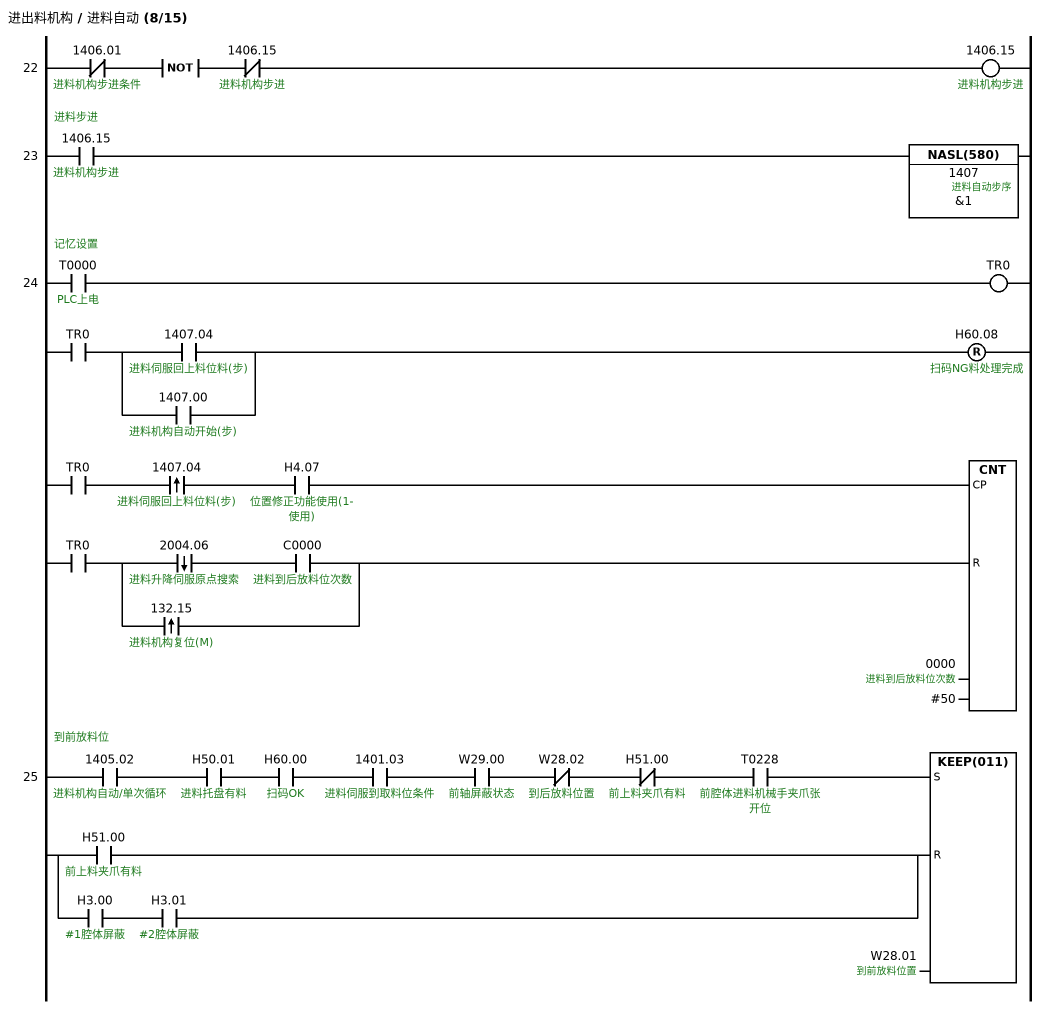
; rung 22
LDNOT 1406.01  ; 进料机构步进条件
NOT(520)
ANDNOT 1406.15  ; 进料机构步进
OUT 1406.15  ; 进料机构步进
; rung 23: 进料步进
LD 1406.15  ; 进料机构步进
NASL(580) 1407 &1  ; 进料自动步序
; rung 24: 记忆设置
LD T0000  ; PLC上电
OUT TR0
LD 1407.04  ; 进料伺服回上料位料(步)
OR 1407.00  ; 进料机构自动开始(步)
ANDLD
RSET H60.08  ; 扫码NG料处理完成
LD TR0
@AND 1407.04  ; 进料伺服回上料位料(步)
AND H4.07  ; 位置修正功能使用(1-使用)
LD TR0
%LD 2004.06  ; 进料升降伺服原点搜索
AND C0000  ; 进料到后放料位次数
@OR 132.15  ; 进料机构复位(M)
ANDLD
CNT 0000 #50  ; 进料到后放料位次数
; rung 25: 到前放料位
LD 1405.02  ; 进料机构自动/单次循环
AND H50.01  ; 进料托盘有料
AND H60.00  ; 扫码OK
AND 1401.03  ; 进料伺服到取料位条件
AND W29.00  ; 前轴屏蔽状态
ANDNOT W28.02  ; 到后放料位置
ANDNOT H51.00  ; 前上料夹爪有料
AND T0228  ; 前腔体进料机械手夹爪张开位
LD H51.00  ; 前上料夹爪有料
LD H3.00  ; #1腔体屏蔽
AND H3.01  ; #2腔体屏蔽
ORLD
KEEP(011) W28.01  ; 到前放料位置

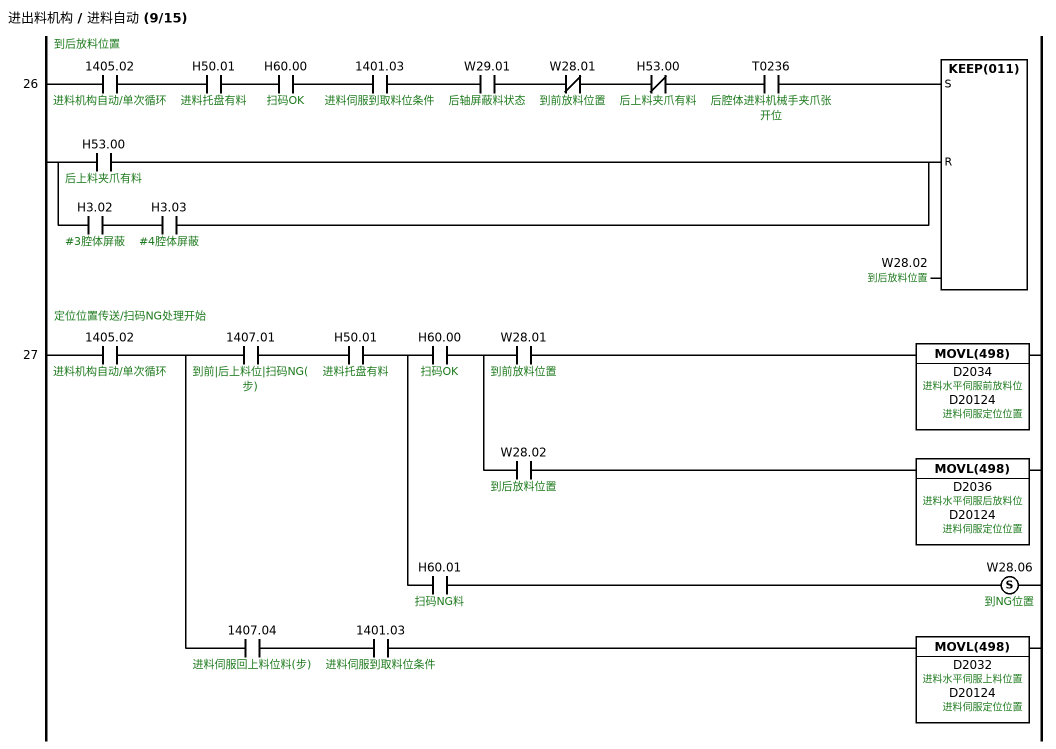
; rung 26: 到后放料位置
LD 1405.02  ; 进料机构自动/单次循环
AND H50.01  ; 进料托盘有料
AND H60.00  ; 扫码OK
AND 1401.03  ; 进料伺服到取料位条件
AND W29.01  ; 后轴屏蔽料状态
ANDNOT W28.01  ; 到前放料位置
ANDNOT H53.00  ; 后上料夹爪有料
AND T0236  ; 后腔体进料机械手夹爪张开位
LD H53.00  ; 后上料夹爪有料
LD H3.02  ; #3腔体屏蔽
AND H3.03  ; #4腔体屏蔽
ORLD
KEEP(011) W28.02  ; 到后放料位置
; rung 27: 定位位置传送/扫码NG处理开始
LD 1405.02  ; 进料机构自动/单次循环
OUT TR0
AND 1407.01  ; 到前|后上料位|扫码NG(步)
AND H50.01  ; 进料托盘有料
OUT TR1
AND H60.00  ; 扫码OK
OUT TR2
AND W28.01  ; 到前放料位置
MOVL(498) D2034 D20124  ; 进料水平伺服前放料位, 进料伺服定位位置
LD TR2
AND W28.02  ; 到后放料位置
MOVL(498) D2036 D20124  ; 进料水平伺服后放料位, 进料伺服定位位置
LD TR1
AND H60.01  ; 扫码NG料
SET W28.06  ; 到NG位置
LD TR0
AND 1407.04  ; 进料伺服回上料位料(步)
AND 1401.03  ; 进料伺服到取料位条件
MOVL(498) D2032 D20124  ; 进料水平伺服上料位置, 进料伺服定位位置

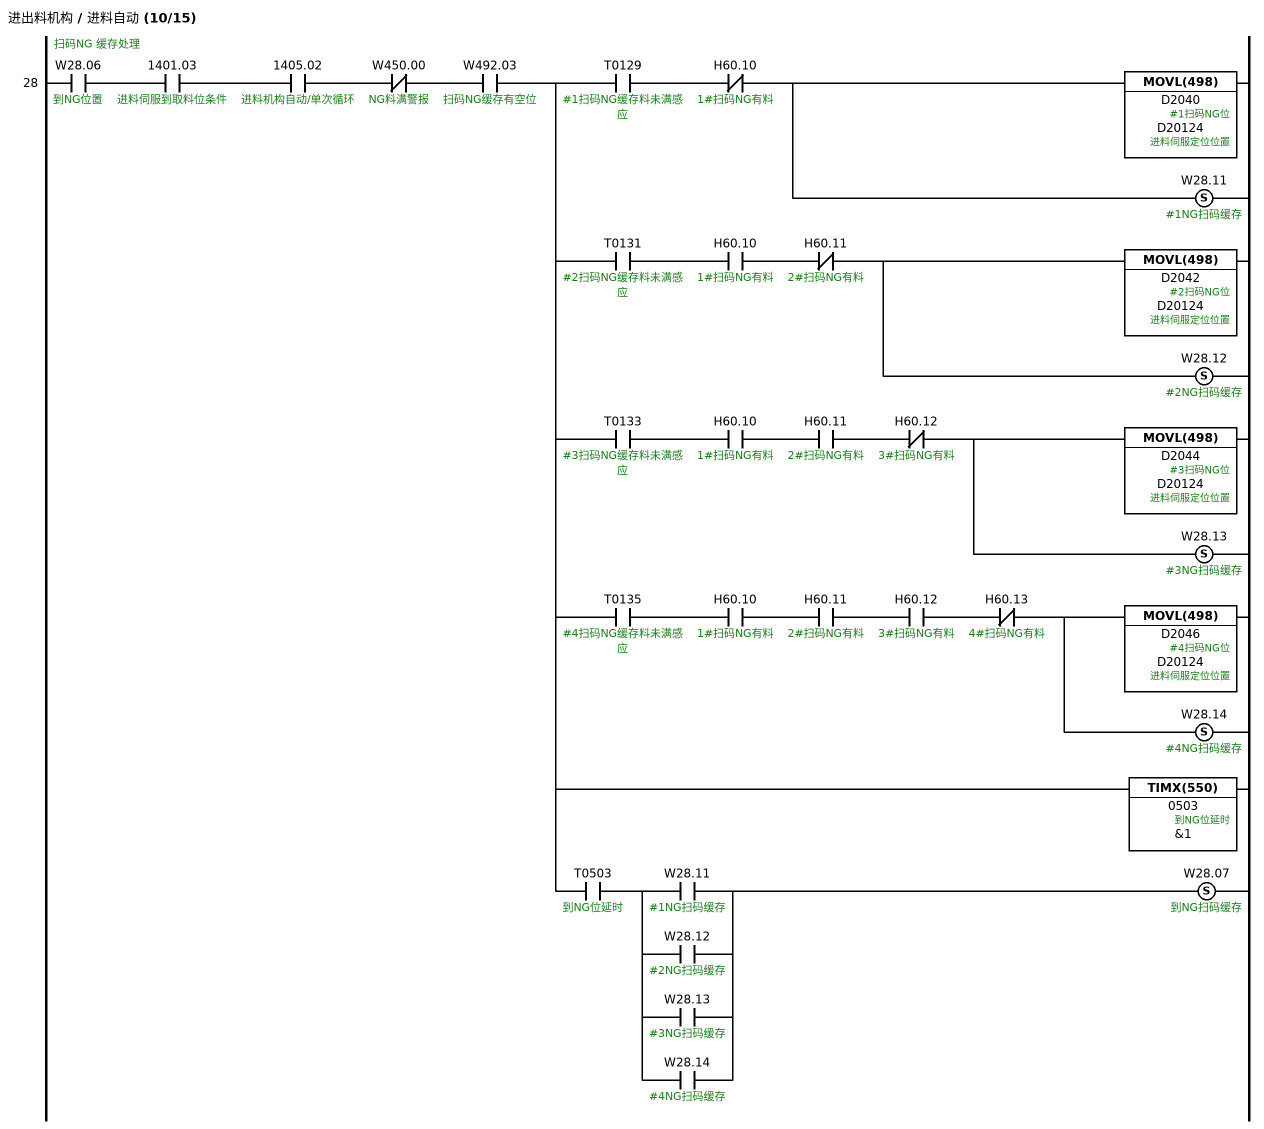
; rung 28: 扫码NG 缓存处理
LD W28.06  ; 到NG位置
AND 1401.03  ; 进料伺服到取料位条件
AND 1405.02  ; 进料机构自动/单次循环
ANDNOT W450.00  ; NG料满警报
AND W492.03  ; 扫码NG缓存有空位
OUT TR0
AND T0129  ; #1扫码NG缓存料未满感应
ANDNOT H60.10  ; 1#扫码NG有料
MOVL(498) D2040 D20124  ; #1扫码NG位, 进料伺服定位位置
SET W28.11  ; #1NG扫码缓存
LD TR0
AND T0131  ; #2扫码NG缓存料未满感应
AND H60.10  ; 1#扫码NG有料
ANDNOT H60.11  ; 2#扫码NG有料
MOVL(498) D2042 D20124  ; #2扫码NG位, 进料伺服定位位置
SET W28.12  ; #2NG扫码缓存
LD TR0
AND T0133  ; #3扫码NG缓存料未满感应
AND H60.10  ; 1#扫码NG有料
AND H60.11  ; 2#扫码NG有料
ANDNOT H60.12  ; 3#扫码NG有料
MOVL(498) D2044 D20124  ; #3扫码NG位, 进料伺服定位位置
SET W28.13  ; #3NG扫码缓存
LD TR0
AND T0135  ; #4扫码NG缓存料未满感应
AND H60.10  ; 1#扫码NG有料
AND H60.11  ; 2#扫码NG有料
AND H60.12  ; 3#扫码NG有料
ANDNOT H60.13  ; 4#扫码NG有料
MOVL(498) D2046 D20124  ; #4扫码NG位, 进料伺服定位位置
SET W28.14  ; #4NG扫码缓存
LD TR0
TIMX(550) 0503 &1  ; 到NG位延时
AND T0503  ; 到NG位延时
LD W28.11  ; #1NG扫码缓存
OR W28.12  ; #2NG扫码缓存
OR W28.13  ; #3NG扫码缓存
OR W28.14  ; #4NG扫码缓存
ANDLD
SET W28.07  ; 到NG扫码缓存

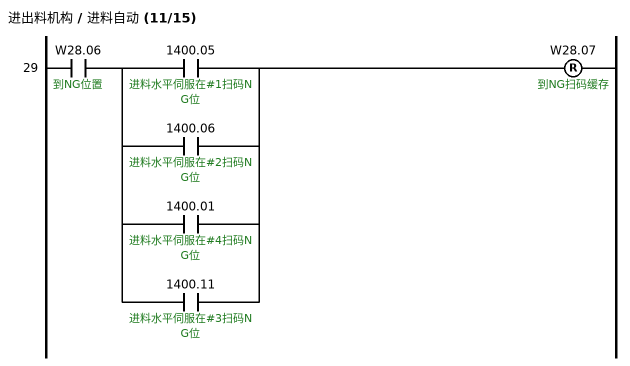
; rung 29
LD W28.06  ; 到NG位置
LD 1400.05  ; 进料水平伺服在#1扫码NG位
OR 1400.06  ; 进料水平伺服在#2扫码NG位
OR 1400.01  ; 进料水平伺服在#4扫码NG位
OR 1400.11  ; 进料水平伺服在#3扫码NG位
ANDLD
RSET W28.07  ; 到NG扫码缓存

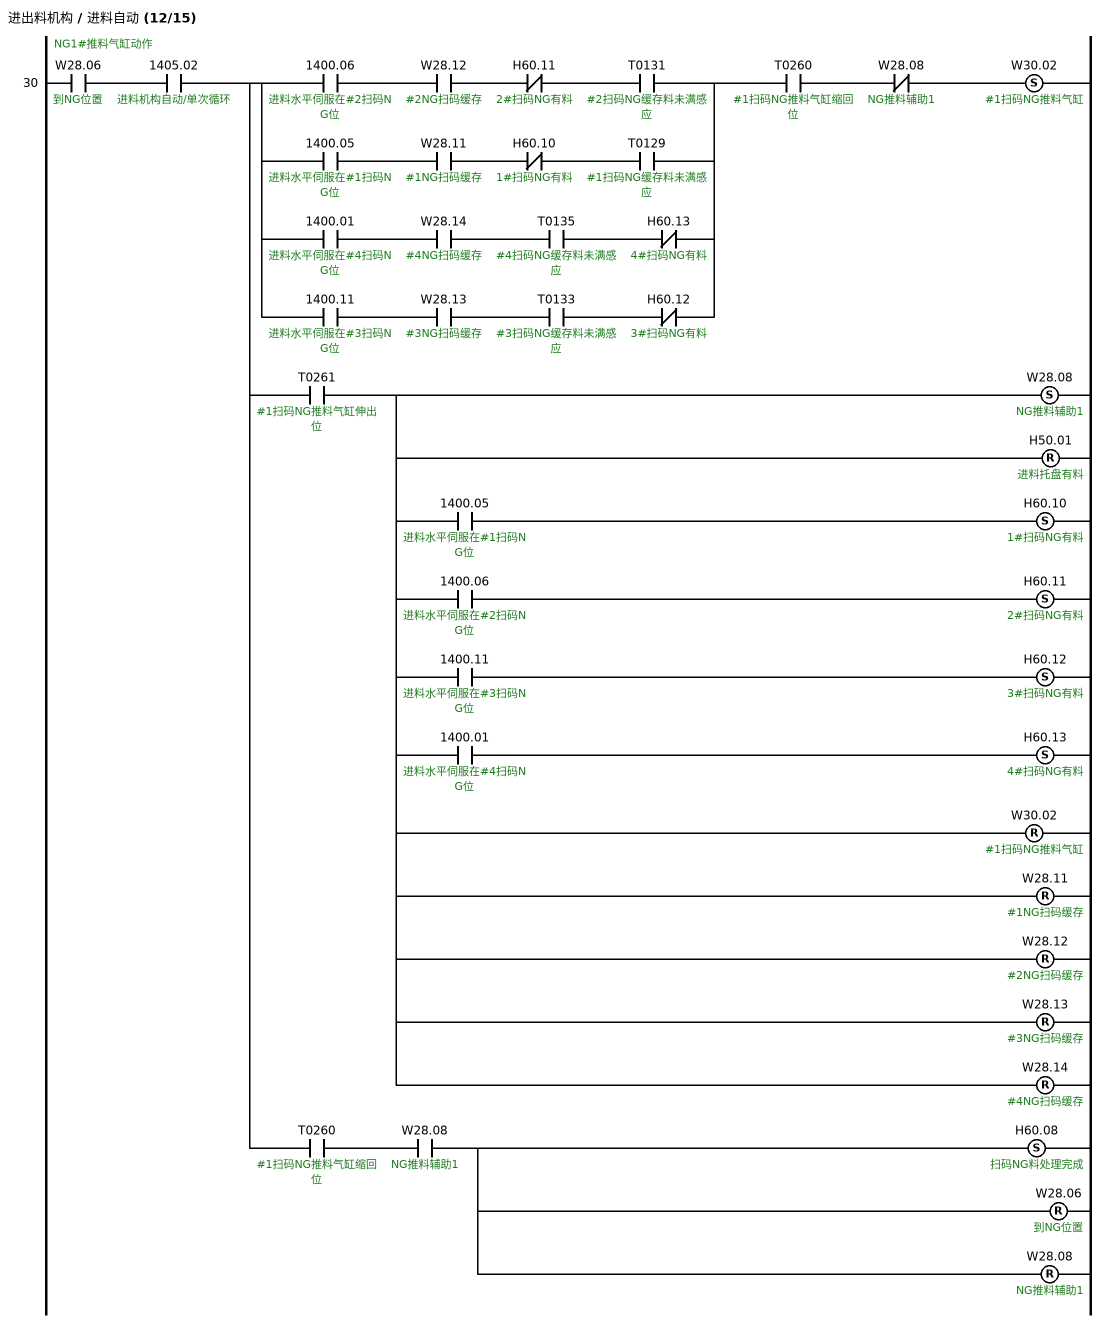
; rung 30: NG1#推料气缸动作
LD W28.06  ; 到NG位置
AND 1405.02  ; 进料机构自动/单次循环
OUT TR0
LD 1400.06  ; 进料水平伺服在#2扫码NG位
AND W28.12  ; #2NG扫码缓存
ANDNOT H60.11  ; 2#扫码NG有料
AND T0131  ; #2扫码NG缓存料未满感应
LD 1400.05  ; 进料水平伺服在#1扫码NG位
AND W28.11  ; #1NG扫码缓存
ANDNOT H60.10  ; 1#扫码NG有料
AND T0129  ; #1扫码NG缓存料未满感应
ORLD
LD 1400.01  ; 进料水平伺服在#4扫码NG位
AND W28.14  ; #4NG扫码缓存
AND T0135  ; #4扫码NG缓存料未满感应
ANDNOT H60.13  ; 4#扫码NG有料
ORLD
LD 1400.11  ; 进料水平伺服在#3扫码NG位
AND W28.13  ; #3NG扫码缓存
AND T0133  ; #3扫码NG缓存料未满感应
ANDNOT H60.12  ; 3#扫码NG有料
ORLD
ANDLD
AND T0260  ; #1扫码NG推料气缸缩回位
ANDNOT W28.08  ; NG推料辅助1
SET W30.02  ; #1扫码NG推料气缸
LD TR0
AND T0261  ; #1扫码NG推料气缸伸出位
OUT TR1
SET W28.08  ; NG推料辅助1
RSET H50.01  ; 进料托盘有料
AND 1400.05  ; 进料水平伺服在#1扫码NG位
SET H60.10  ; 1#扫码NG有料
LD TR1
AND 1400.06  ; 进料水平伺服在#2扫码NG位
SET H60.11  ; 2#扫码NG有料
LD TR1
AND 1400.11  ; 进料水平伺服在#3扫码NG位
SET H60.12  ; 3#扫码NG有料
LD TR1
AND 1400.01  ; 进料水平伺服在#4扫码NG位
SET H60.13  ; 4#扫码NG有料
LD TR1
RSET W30.02  ; #1扫码NG推料气缸
RSET W28.11  ; #1NG扫码缓存
RSET W28.12  ; #2NG扫码缓存
RSET W28.13  ; #3NG扫码缓存
RSET W28.14  ; #4NG扫码缓存
LD TR0
AND T0260  ; #1扫码NG推料气缸缩回位
AND W28.08  ; NG推料辅助1
SET H60.08  ; 扫码NG料处理完成
RSET W28.06  ; 到NG位置
RSET W28.08  ; NG推料辅助1

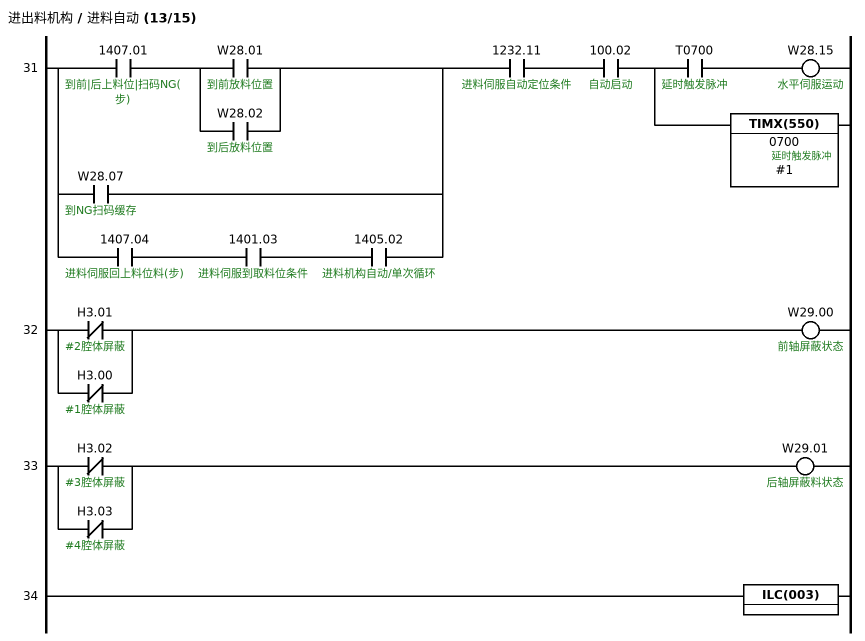
; rung 31
LD 1407.01  ; 到前|后上料位|扫码NG(步)
LD W28.01  ; 到前放料位置
OR W28.02  ; 到后放料位置
ANDLD
OR W28.07  ; 到NG扫码缓存
LD 1407.04  ; 进料伺服回上料位料(步)
AND 1401.03  ; 进料伺服到取料位条件
AND 1405.02  ; 进料机构自动/单次循环
ORLD
AND 1232.11  ; 进料伺服自动定位条件
AND 100.02  ; 自动启动
OUT TR0
AND T0700  ; 延时触发脉冲
OUT W28.15  ; 水平伺服运动
LD TR0
TIMX(550) 0700 #1  ; 延时触发脉冲
; rung 32
LDNOT H3.01  ; #2腔体屏蔽
ORNOT H3.00  ; #1腔体屏蔽
OUT W29.00  ; 前轴屏蔽状态
; rung 33
LDNOT H3.02  ; #3腔体屏蔽
ORNOT H3.03  ; #4腔体屏蔽
OUT W29.01  ; 后轴屏蔽料状态
; rung 34
ILC(003)

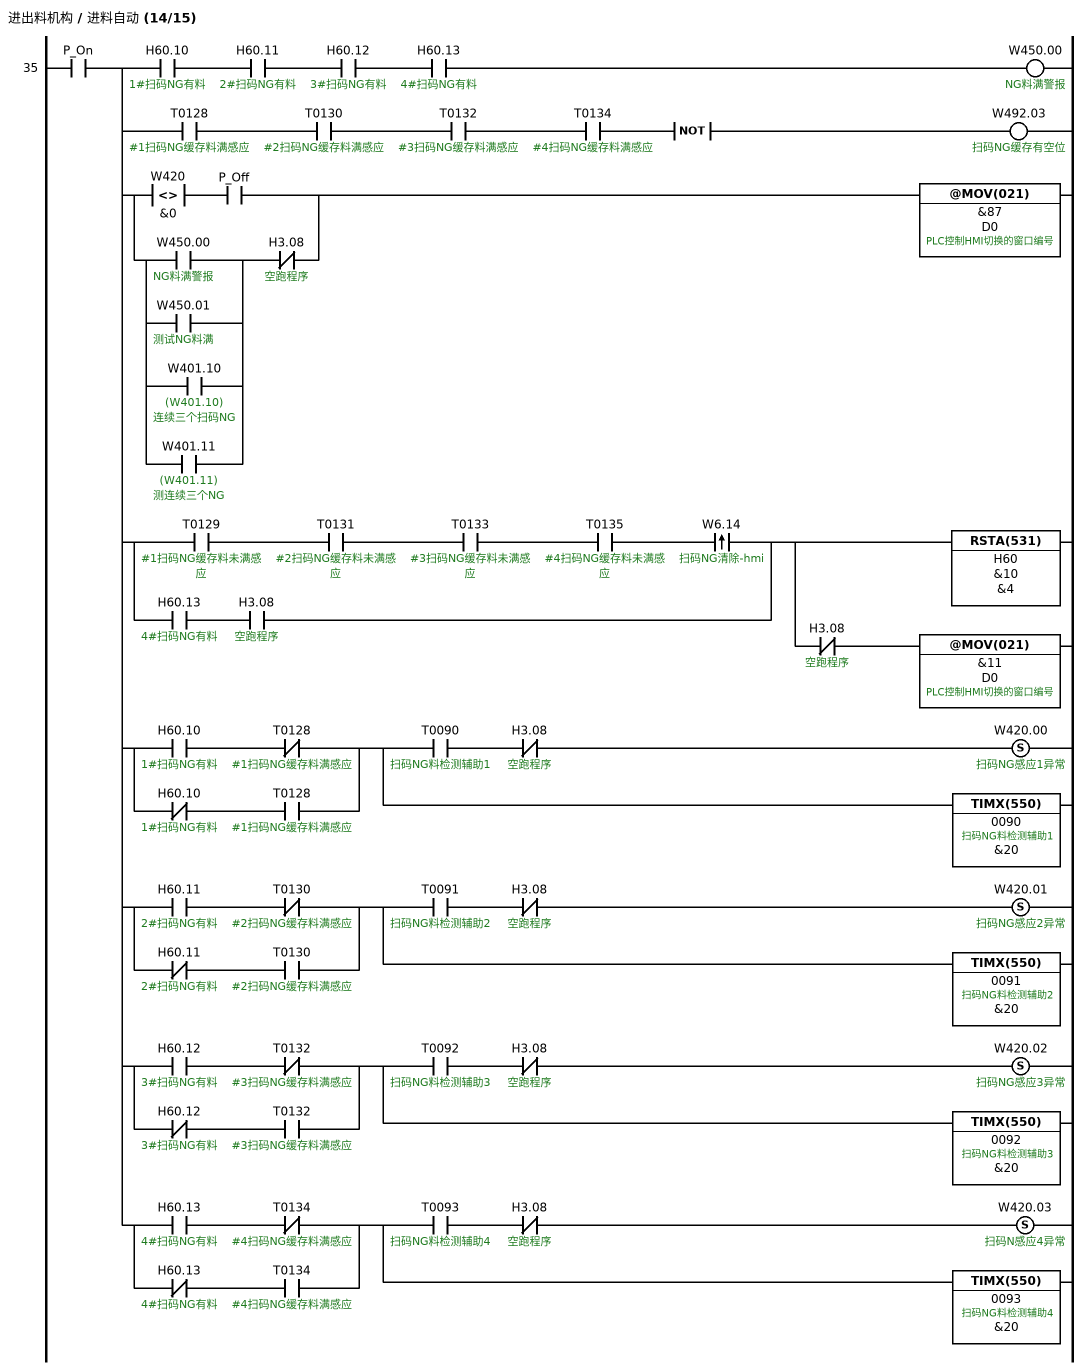
; rung 35
LD P_On
OUT TR0
AND H60.10  ; 1#扫码NG有料
AND H60.11  ; 2#扫码NG有料
AND H60.12  ; 3#扫码NG有料
AND H60.13  ; 4#扫码NG有料
OUT W450.00  ; NG料满警报
LD TR0
AND T0128  ; #1扫码NG缓存料满感应
AND T0130  ; #2扫码NG缓存料满感应
AND T0132  ; #3扫码NG缓存料满感应
AND T0134  ; #4扫码NG缓存料满感应
NOT(520)
OUT W492.03  ; 扫码NG缓存有空位
LD TR0
LD<>(305) W420 &0
AND P_Off
LD W450.00  ; NG料满警报
OR W450.01  ; 测试NG料满
OR W401.10  ; (W401.10) 连续三个扫码NG
OR W401.11  ; (W401.11) 测连续三个NG
ANDNOT H3.08  ; 空跑程序
ORLD
ANDLD
@MOV(021) &87 D0  ; PLC控制HMI切换的窗口编号
LD TR0
LD T0129  ; #1扫码NG缓存料未满感应
AND T0131  ; #2扫码NG缓存料未满感应
AND T0133  ; #3扫码NG缓存料未满感应
AND T0135  ; #4扫码NG缓存料未满感应
@AND W6.14  ; 扫码NG清除-hmi
LD H60.13  ; 4#扫码NG有料
AND H3.08  ; 空跑程序
ORLD
ANDLD
RSTA(531) H60 &10 &4
ANDNOT H3.08  ; 空跑程序
@MOV(021) &11 D0  ; PLC控制HMI切换的窗口编号
LD TR0
LD H60.10  ; 1#扫码NG有料
ANDNOT T0128  ; #1扫码NG缓存料满感应
LDNOT H60.10  ; 1#扫码NG有料
AND T0128  ; #1扫码NG缓存料满感应
ORLD
ANDLD
OUT TR1
AND T0090  ; 扫码NG料检测辅助1
ANDNOT H3.08  ; 空跑程序
SET W420.00  ; 扫码NG感应1异常
LD TR1
TIMX(550) 0090 &20  ; 扫码NG料检测辅助1
LD TR0
LD H60.11  ; 2#扫码NG有料
ANDNOT T0130  ; #2扫码NG缓存料满感应
LDNOT H60.11  ; 2#扫码NG有料
AND T0130  ; #2扫码NG缓存料满感应
ORLD
ANDLD
OUT TR1
AND T0091  ; 扫码NG料检测辅助2
ANDNOT H3.08  ; 空跑程序
SET W420.01  ; 扫码NG感应2异常
LD TR1
TIMX(550) 0091 &20  ; 扫码NG料检测辅助2
LD TR0
LD H60.12  ; 3#扫码NG有料
ANDNOT T0132  ; #3扫码NG缓存料满感应
LDNOT H60.12  ; 3#扫码NG有料
AND T0132  ; #3扫码NG缓存料满感应
ORLD
ANDLD
OUT TR1
AND T0092  ; 扫码NG料检测辅助3
ANDNOT H3.08  ; 空跑程序
SET W420.02  ; 扫码NG感应3异常
LD TR1
TIMX(550) 0092 &20  ; 扫码NG料检测辅助3
LD TR0
LD H60.13  ; 4#扫码NG有料
ANDNOT T0134  ; #4扫码NG缓存料满感应
LDNOT H60.13  ; 4#扫码NG有料
AND T0134  ; #4扫码NG缓存料满感应
ORLD
ANDLD
OUT TR0
AND T0093  ; 扫码NG料检测辅助4
ANDNOT H3.08  ; 空跑程序
SET W420.03  ; 扫码N感应4异常
LD TR0
TIMX(550) 0093 &20  ; 扫码NG料检测辅助4

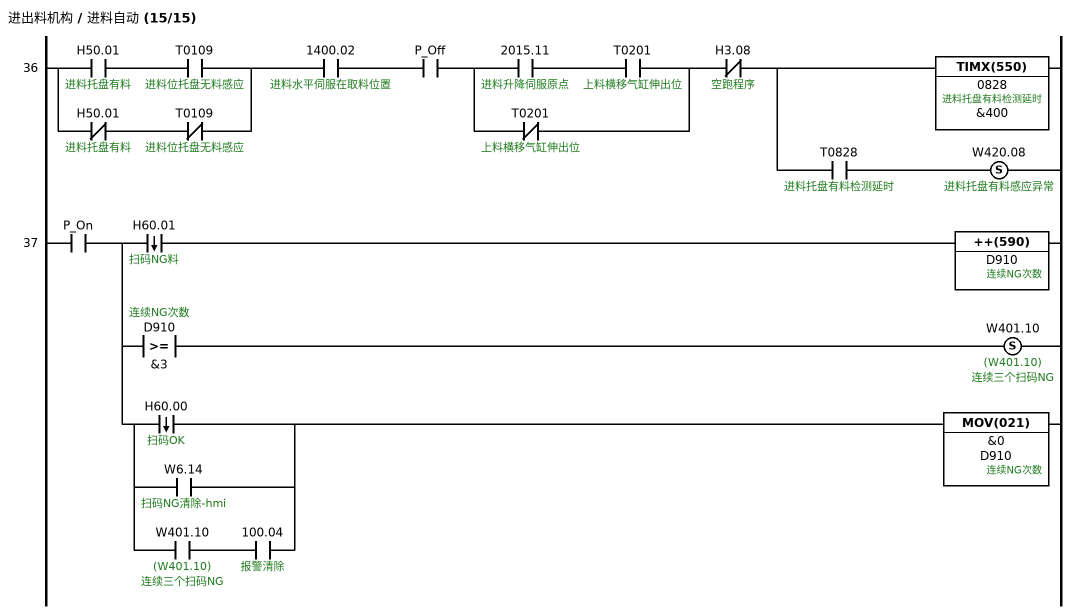
; rung 36
LD H50.01  ; 进料托盘有料
AND T0109  ; 进料位托盘无料感应
LDNOT H50.01  ; 进料托盘有料
ANDNOT T0109  ; 进料位托盘无料感应
ORLD
AND 1400.02  ; 进料水平伺服在取料位置
AND P_Off
LD 2015.11  ; 进料升降伺服原点
AND T0201  ; 上料横移气缸伸出位
ORNOT T0201  ; 上料横移气缸伸出位
ANDLD
ANDNOT H3.08  ; 空跑程序
TIMX(550) 0828 &400  ; 进料托盘有料检测延时
AND T0828  ; 进料托盘有料检测延时
SET W420.08  ; 进料托盘有料感应异常
; rung 37
LD P_On
OUT TR0
%AND H60.01  ; 扫码NG料
++(590) D910  ; 连续NG次数
LD TR0
AND>=(325) D910 &3  ; 连续NG次数
SET W401.10  ; (W401.10) 连续三个扫码NG
LD TR0
%LD H60.00  ; 扫码OK
OR W6.14  ; 扫码NG清除-hmi
LD W401.10  ; (W401.10) 连续三个扫码NG
AND 100.04  ; 报警清除
ORLD
ANDLD
MOV(021) &0 D910  ; 连续NG次数

### Section 出料手动

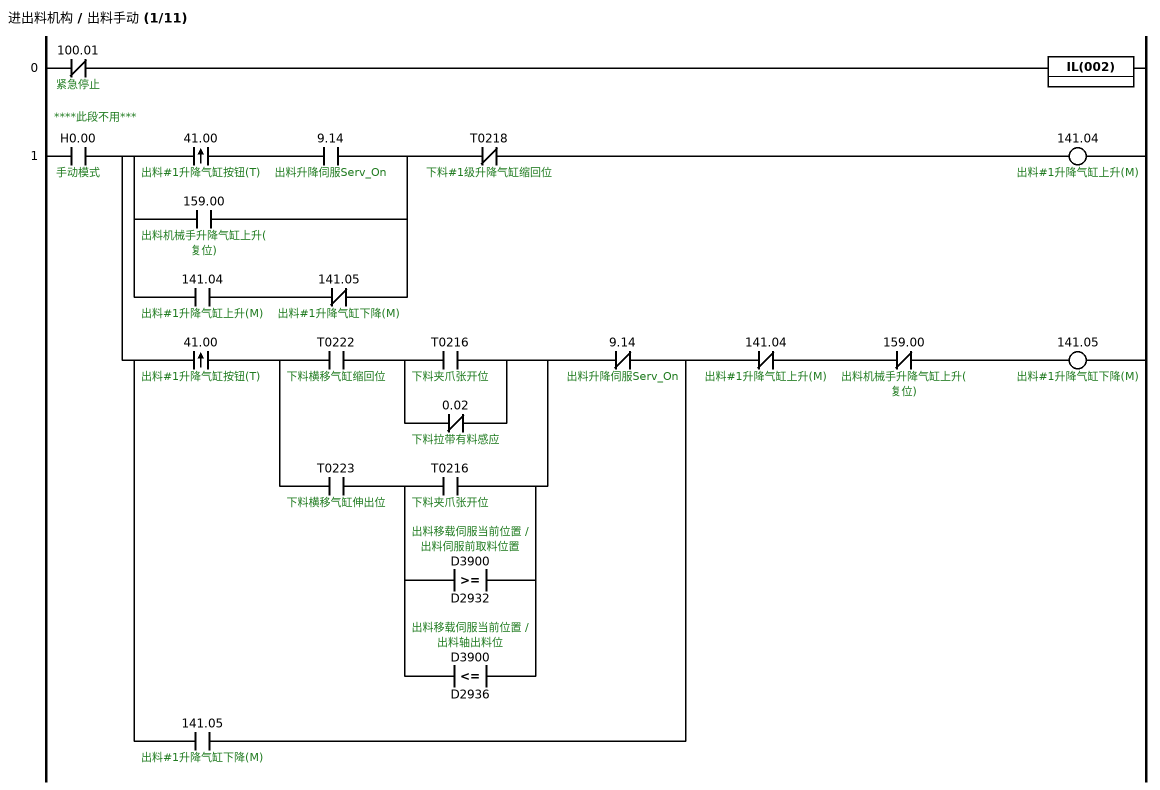
; rung 0
LDNOT 100.01  ; 紧急停止
IL(002)
; rung 1: ****此段不用***
LD H0.00  ; 手动模式
OUT TR0
@LD 41.00  ; 出料#1升降气缸按钮(T)
AND 9.14  ; 出料升降伺服Serv_On
OR 159.00  ; 出料机械手升降气缸上升(复位)
LD 141.04  ; 出料#1升降气缸上升(M)
ANDNOT 141.05  ; 出料#1升降气缸下降(M)
ORLD
ANDLD
ANDNOT T0218  ; 下料#1级升降气缸缩回位
OUT 141.04  ; 出料#1升降气缸上升(M)
LD TR0
@LD 41.00  ; 出料#1升降气缸按钮(T)
LD T0222  ; 下料横移气缸缩回位
LD T0216  ; 下料夹爪张开位
ORNOT 0.02  ; 下料拉带有料感应
ANDLD
LD T0223  ; 下料横移气缸伸出位
LD T0216  ; 下料夹爪张开位
OR>=SL(328) D3900 D2932  ; 出料移载伺服当前位置, 出料伺服前取料位置
OR<=SL(318) D3900 D2936  ; 出料移载伺服当前位置, 出料轴出料位
ANDLD
ORLD
ANDLD
ANDNOT 9.14  ; 出料升降伺服Serv_On
OR 141.05  ; 出料#1升降气缸下降(M)
ANDLD
ANDNOT 141.04  ; 出料#1升降气缸上升(M)
ANDNOT 159.00  ; 出料机械手升降气缸上升(复位)
OUT 141.05  ; 出料#1升降气缸下降(M)

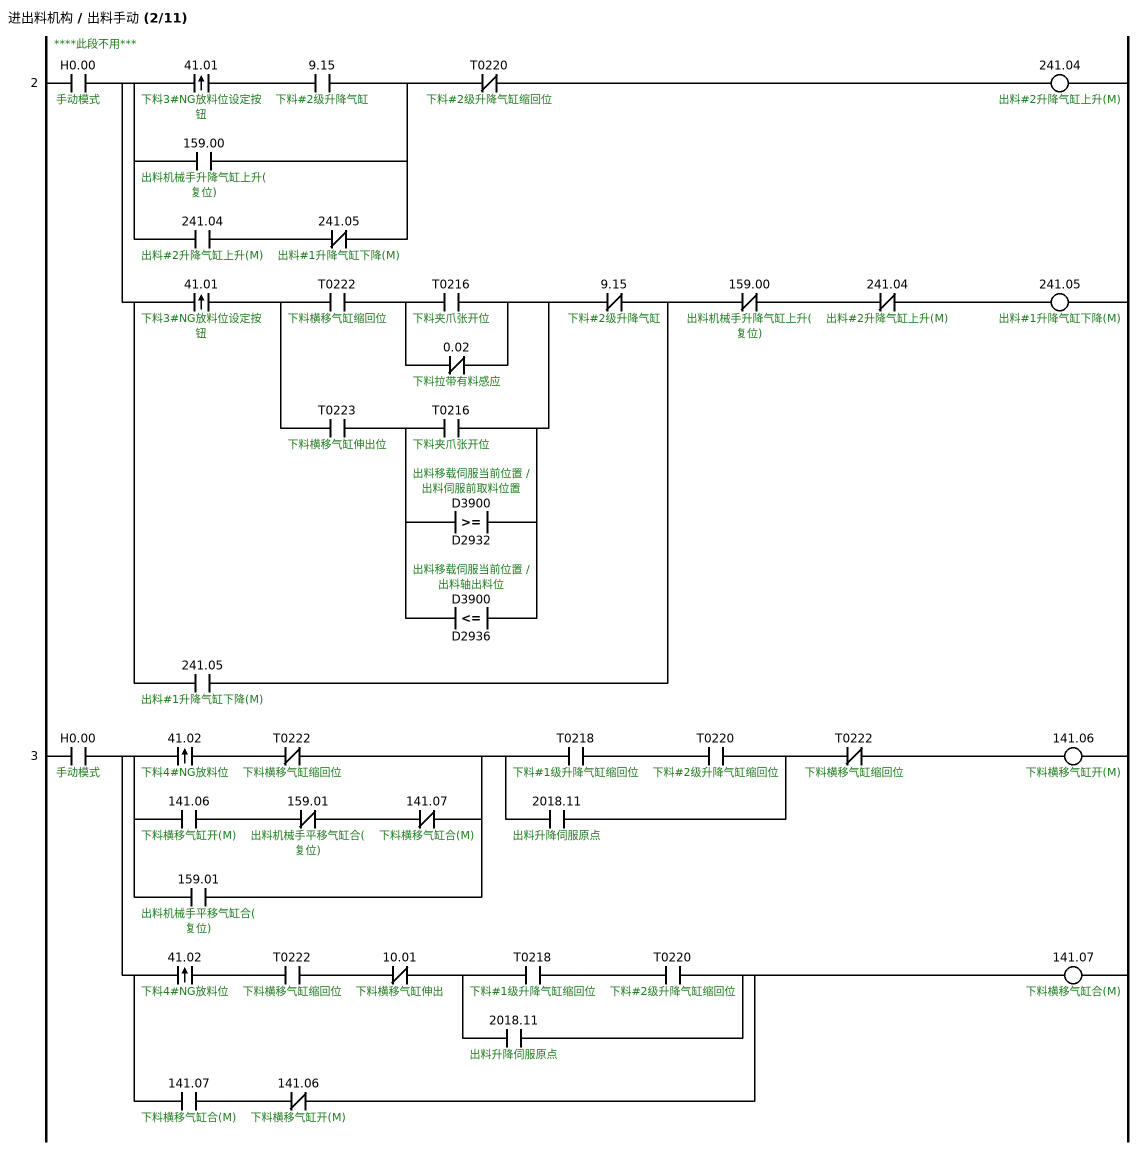
; rung 2: ****此段不用***
LD H0.00  ; 手动模式
OUT TR0
@LD 41.01  ; 下料3#NG放料位设定按钮
AND 9.15  ; 下料#2级升降气缸
OR 159.00  ; 出料机械手升降气缸上升(复位)
LD 241.04  ; 出料#2升降气缸上升(M)
ANDNOT 241.05  ; 出料#1升降气缸下降(M)
ORLD
ANDLD
ANDNOT T0220  ; 下料#2级升降气缸缩回位
OUT 241.04  ; 出料#2升降气缸上升(M)
LD TR0
@LD 41.01  ; 下料3#NG放料位设定按钮
LD T0222  ; 下料横移气缸缩回位
LD T0216  ; 下料夹爪张开位
ORNOT 0.02  ; 下料拉带有料感应
ANDLD
LD T0223  ; 下料横移气缸伸出位
LD T0216  ; 下料夹爪张开位
OR>=SL(328) D3900 D2932  ; 出料移载伺服当前位置, 出料伺服前取料位置
OR<=SL(318) D3900 D2936  ; 出料移载伺服当前位置, 出料轴出料位
ANDLD
ORLD
ANDLD
ANDNOT 9.15  ; 下料#2级升降气缸
OR 241.05  ; 出料#1升降气缸下降(M)
ANDLD
ANDNOT 159.00  ; 出料机械手升降气缸上升(复位)
ANDNOT 241.04  ; 出料#2升降气缸上升(M)
OUT 241.05  ; 出料#1升降气缸下降(M)
; rung 3
LD H0.00  ; 手动模式
OUT TR0
@LD 41.02  ; 下料4#NG放料位
ANDNOT T0222  ; 下料横移气缸缩回位
LD 141.06  ; 下料横移气缸开(M)
ANDNOT 159.01  ; 出料机械手平移气缸合(复位)
ANDNOT 141.07  ; 下料横移气缸合(M)
ORLD
OR 159.01  ; 出料机械手平移气缸合(复位)
ANDLD
LD T0218  ; 下料#1级升降气缸缩回位
AND T0220  ; 下料#2级升降气缸缩回位
OR 2018.11  ; 出料升降伺服原点
ANDLD
ANDNOT T0222  ; 下料横移气缸缩回位
OUT 141.06  ; 下料横移气缸开(M)
LD TR0
@LD 41.02  ; 下料4#NG放料位
AND T0222  ; 下料横移气缸缩回位
ANDNOT 10.01  ; 下料横移气缸伸出
LD T0218  ; 下料#1级升降气缸缩回位
AND T0220  ; 下料#2级升降气缸缩回位
OR 2018.11  ; 出料升降伺服原点
ANDLD
LD 141.07  ; 下料横移气缸合(M)
ANDNOT 141.06  ; 下料横移气缸开(M)
ORLD
ANDLD
OUT 141.07  ; 下料横移气缸合(M)

